(* POU XTEST/Baustein Tests/control_test, CFC *)
PROGRAM control_test
VAR
	Offset : REAL;
	x1: FT_PT1;
	step: REAL;
	t1: TIME := T#1s;
	Out: REAL;
	x2: FT_PT2;
	d: REAL := 0.5;
	out2: REAL;
	x3: FT_PID;
	TV, TN : REAL := 1;
	out3: REAL;
	SET: REAL;
	x4: FT_PI;
	M_in: REAL;
	M_en: BOOL;
	RST: BOOL;
	INTB: REAL := 10;
	KP: REAL := 1;
	KI: REAL := 1;
	L_L: REAL := -1000;
	L_H: REAL := 1000;
	out4: REAL;
	l1: BOOL;
	o1: BOOL;
	l2: BOOL;
	o2: BOOL;
	x5: FT_PT1;
END_VAR
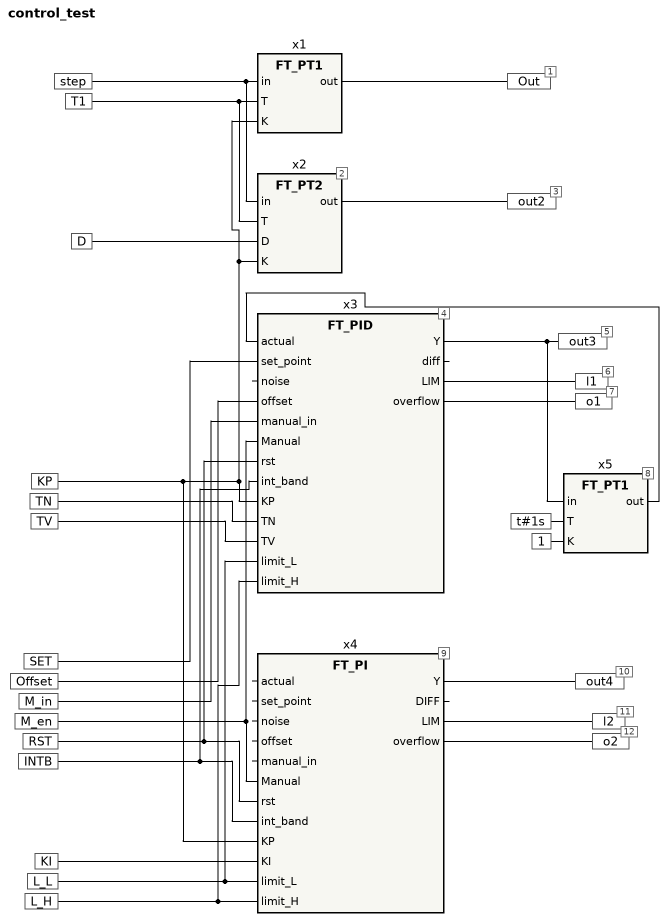
_CFC_ (* Continuous Function Chart, elements in execution order *)
#0 x1:FT_PT1(in: step, T: T1, K: KP)
#1 Out <= #0.out
#2 x2:FT_PT2(in: step, T: T1, D: D, K: KP)
#3 out2 <= #2.out
#4 x3:FT_PID(actual: #8.out, set_point: SET, noise: -, offset: Offset, manual_in: M_in, Manual: M_en, rst: RST, int_band: INTB, KP: KP, TN: TN, TV: TV, limit_L: L_L, limit_H: L_H)
#5 out3 <= #4.Y
#6 l1 <= #4.LIM
#7 o1 <= #4.overflow
#8 x5:FT_PT1(in: #4.Y, T: t#1s, K: 1)
#9 x4:FT_PI(actual: -, set_point: -, noise: -, offset: -, manual_in: -, Manual: M_en, rst: RST, int_band: INTB, KP: KP, KI: KI, limit_L: L_L, limit_H: L_H)
#10 out4 <= #9.Y
#11 l2 <= #9.LIM
#12 o2 <= #9.overflow
_END_CFC_
(* the same logic as Structured Text *)
x1(in := step, T := T1, K := KP);
Out := x1.out;
x2(in := step, T := T1, D := D, K := KP);
out2 := x2.out;
x3(actual := x5.out, set_point := SET, offset := Offset, manual_in := M_in, Manual := M_en, rst := RST, int_band := INTB, KP := KP, TN := TN, TV := TV, limit_L := L_L, limit_H := L_H);
out3 := x3.Y;
l1 := x3.LIM;
o1 := x3.overflow;
x5(in := x3.Y, T := t#1s, K := 1);
x4(Manual := M_en, rst := RST, int_band := INTB, KP := KP, KI := KI, limit_L := L_L, limit_H := L_H);
out4 := x4.Y;
l2 := x4.LIM;
o2 := x4.overflow;
END_PROGRAM

(* POU Engineering/control/FT_PT1, ST *)
FUNCTION_BLOCK FT_PT1
VAR_INPUT
	in : REAL;
	T : TIME;
	K : REAL := 1;
END_VAR
VAR_OUTPUT
	out : REAL;
END_VAR
VAR
	last : DWORD;
	tx: DWORD;
	init: BOOL;
END_VAR

(*
version 1.7	5 jan 2008
programmer 	hugo
tested by		tobias

FT_PT1 is an low pass filter with a programmable time T and faktor K.
 
*)
(* read system time *)
tx := T_PLC_US();

(* startup initialisation *)
IF NOT init THEN
	last := tx;
	init := TRUE;
	out := K * in;
ELSIF T = t#0s THEN
	out := K * in;
ELSE
	out := out + (in * K - out) * (Tx - last) / TIME_TO_REAL(T) * 1E-3;
END_IF;
last := tx;

(*
hm 1.1.2007	rev 1.1
	corrected error while startup value was not correct
	for very small time values real output would run out of range.

hm 3.1.2007	rev 1.2
	corrected an error for falling edge failures.
	added output faktor K.

hm 27. 2. 2007	rev 1.3
	output will be input during init for definitive startup condition.

hm	15.9.2007	rev 1.4
	changed time() to T_PLC_US() for compatibilitxy resons
	increased internal accuracy to Microseconds instead of Milliseconds

hm	23. oct 2007	rev 1.5
	added out := in to the init statements

hm	30. nov 2007	rev 1.6
	changed out to be K * in during initialization

hm	5. jan 2008		rev 1.7
	improved code for better performance
*)
END_FUNCTION_BLOCK

(* POU Engineering/measurements/T_PLC_US, ST *)
FUNCTION T_PLC_US : DWORD
VAR CONSTANT
	debug : BOOL := FALSE;
	N : INT := 0;
	offset : DWORD := 0;
END_VAR
VAR
	tx : TIME;
	temp : DWORD := 1;
END_VAR

(*
version 1.1	12 nov 2007
programmer 	hugo
tested by		tobias

T_PLC_US reads the internal PLC timer and return the time, it has the advantage to be able to set a debug mode 
and speed up the counter to test the plc timer overrun which occurs every 50 days respectively 25 days at siemens S7
this routine also allows to correct the behavior of s7 where the internal plc counter will not count all 32 bits.

*)
tx := TIME();
T_PLC_US := TIME_TO_DWORD(Tx)*1000;
(* hier muss die korrektur für step7 stattfinden
plctime muss den vollen wertebereich von time ausnutzen:
wenn bei step7 time -24tage bis plus 24 tage ist dann muss der timer auch beim überlauf auf -24tage springen 
und auf keinen fall auf 0 !!!!
für siemens muss ein weiterer fb im main eingebunden werden der sicherstellt das alle 32 bits durchgezählt werden.
es kann nur ein fb sein den er muss sich das oberste (32te) bit merken.
oder etwa spring s7 bei überlauf auf -24 tage????? dann wäre keine korrektur nötig.
*)
IF debug THEN
	T_PLC_US := (SHL(T_PLC_US,N) OR SHL(temp,N)-1) + Offset;
END_IF;

(* revision history
hm	14.9.2007	rev 1.0
	original version

hm	12. nov 2007	rev 1.1
	added temporaray variable tx because some compilers could not handle time() as an argument

*)
END_FUNCTION

(* POU Engineering/control/FT_PT2, ST *)
FUNCTION_BLOCK FT_PT2
VAR_INPUT
	in : REAL;
	T : TIME;
	D : REAL;
	K : REAL := 1;
END_VAR
VAR_OUTPUT
	out : REAL;
END_VAR
VAR
	init: BOOL;
	int1 : FT_INT;
	int2 : FT_INT;
	tn: REAL;
END_VAR

(*
version 1.3	30 Nov 2007
programmer 	hugo
tested by		tobias

FT_PT2 is a 2nd grade filter with programmable times T, D and faktor K.
 
*)
(* startup initialisation *)
IF NOT init THEN
	out := K * in;
	init := TRUE;
ELSIF T = t#0s THEN
	out := K * in;
ELSE
	tn := TIME_TO_REAL(T)/1000;
	int1(in := in * K / (TN * TN) - int1.Out * 2 *D / TN - int2.Out / (TN * TN));
	int2(in := int1.Out);
	out := int2.out;
END_IF;

(* revision history

15.1.2007 hm		rev 1.1
	changed formula to new more acurate formula
	old code:
	tx := TIME();
	IF NOT init THEN
		last := tx;
		init := TRUE;
	ELSE
		IF T> t#0s THEN
			out1 := out1 + (in - out1) * TIME_TO_REAL(Tx - last) / TIME_TO_REAL(T);
		ELSE
			out1 := in;
		END_IF;
		IF T > t#0s THEN
			out2 := out2 + (out1 - out2) * TIME_TO_REAL(Tx - last) / TIME_TO_REAL(T);
		ELSE
			out2 := out1;
		END_IF;
		out := out2 * K;
	END_IF;
	last := tx;

hm 		15.9.2007		rev 1.2
	deleted unused code for init system time reading tx	

hm		30.11.2007		rev 1.3
	changed out to be K * in during initialization
	avoind divide by 0 if tn = 0
*)
END_FUNCTION_BLOCK

(* POU Engineering/control/FT_INT, ST *)
FUNCTION_BLOCK FT_INT
VAR_INPUT
	in : REAL;
	K : REAL := 1;
	run : BOOL := 1;
	rst: BOOL := 0;
	out_min : REAL := -1E37;
	out_max : REAL := 1E37;
END_VAR
VAR_OUTPUT
	Out : REAL;
END_VAR
VAR
	last: DWORD;
	in_last : REAL;
	tx: DWORD;
	init: BOOL;
	tc: DWORD;
	out1: REAL;
	out2: REAL;
END_VAR


(*
version 1.8	13. mar 2008
programmer 	hugo
tested by		tobias

FT_int is an integrator with input IN and factor K.
integration is only done while run = true, if run is false integration is stopped and the out remains at the last value.
if run is left unconnected, run is considered true by the function block.
the output ET will display the total integration time from last reset.
a rst input will reset output and the timer ET to 0.
the out_min and out_max values can be set to ,imit the output value range. 
the default for K is 1.

 
*)
(* read and store system time *)
tx := T_PLC_US();
tc := tx - last;

(* startup initialisation *)
IF rst OR NOT init THEN
	out1 := 0;
	out2 := 0;
	init := TRUE;
	last := tx;
ELSIF run AND tc > 0 THEN
	last := tx;
	out1 := out1 + (in + in_last) * tc * K * 5E-7;
	IF ABS(out1) > ABS(out2) THEN
		out2 := out2 + out1;
		out1:= 0;
	END_IF;
ELSIF NOT run THEN
	last := tx;
END_IF;
in_last := in;
out := out1 + out2;
IF out > out_max THEN
	out2 := out_max;
	out1 := 0;
	out := out_max;
ELSIF out < out_min THEN
	out2 := out_min;
	out1 := 0;
	out := out_min;
END_IF;


(*
hm 13.12.2006	rev 1.1
	changed to "trapezregel" which increases accuracy
	before out := out + in * time new: out := out + (in + in_last) / 2 * time

hm 15.1.2007		rev 1.2
	added default for k to be 1.

hm	15.9.2007		rev 1.3
	replaced time() with T_PLC_US for compatibility and performance reason
	increased internal accuracy to microseconds

hm 29. oct 2007		rev 1.4
	changed code so int will not be called is time difference is 0 to increase accuracy on systems
	with cycle times below 1ms

hm	2. dec 2007	 	rev 1.5
	changed code for better performance

hm	5. jan 2008		rev 1.6
	further improvements in performance

hm	8. feb 2008		rev 1.7
	deleted limits +/- 1000 now limit is the range of real
	added variables out1 and out2 to extend the resolution
	corrected an error with elapsed time
	deleted unusfull output ET

hm	13. mar 2008		rev 1.8
	changed preset value out_min to -1e37.
	stop integrator at the limits.
*)
END_FUNCTION_BLOCK

(* POU Engineering/control/FT_PID, ST *)
FUNCTION_BLOCK FT_PID
VAR_INPUT
	actual, set_point, noise, offset, manual_in : REAL;
	Manual : BOOL;
	rst : BOOL := FALSE;
	int_band : REAL := 100;
	KP : REAL := 1.0;
	TN : REAL := 1.0;
	TV : REAL := 1.0;
	limit_L : REAL := -1000;
	limit_H : REAL := 1000;
END_VAR
VAR_INPUT CONSTANT
	int_limit_L : REAL := -1000;
	int_limit_H : REAL := 1000;
END_VAR
VAR_OUTPUT
	Y : REAL;
	diff: REAL;
	LIM, overflow : BOOL;
END_VAR
VAR
	integ : FT_INT;
	deriv : FT_deriv;
END_VAR

(*
version 1.6	5 jan 2008
programmer 	hugo
tested by		tobias

FT_PID is a pid controller with manual functionality.
The PID controller works according to the fomula Y = KP * ( e + 1/TN * INTEG(e) + TV *DERIV(e)) + offset, while e = set_point - actual.
a rst will reset all internal data, while a switch to manual will cause the controller to follow the function Y = manual_in + offset.
limit_h and Limit_l set the possible output range of Y.
the output flags lim will signal that the output limits are active and overflow will signal that the integrator has reached the max or min limit.  

since rev 1.1 the "trapezregel is used for more accuracy.
rev 1.2 added selective integratin which means the integrative component is only active within a small range of the target value 
this avoids the integrator to go to limits while an input setpoint change happened and is only causing overshoots.
the int_band is by default 100 which means the int is active all the time and if set to for example to 0.1 the integrator is only active
while the input is between 0.9 and 1.1 of the set_point value.

default values for KP = 1, TN = 1, TV = 1, LIMIT_L = -1000, LIMIT_H = +1000.
*)
IF NOT rst AND NOT manual THEN
	(* calculate the process error *)
	DIFF := DEAD_BAND(set_point - actual, Noise);
	IF ABS(diff) <= int_band AND NOT overflow AND TN > 0 THEN
		(* integrator is within int_band and needs to be run *)
		integ(in := diff, K := 1/TN, run := TRUE, rst := FALSE, out_min := int_limit_L, out_max := int_limit_H);
		(* check if integrator has reached its limits and set overflow *)
		IF integ.Out >= int_limit_H OR integ.Out <= int_limit_L THEN overflow := TRUE; END_IF;
	ELSE
		(* int_band is exceeded, integrator needs to be cleared *)
		integ(rst := TRUE);
	END_IF;
	(* calculate the derivative part *)
	deriv(in := diff, K := TV);
	(* add up all parts *)
	Y := KP * (integ.Out + deriv.out + diff);
ELSIF rst THEN
	integ(rst := TRUE);		(* reset the integrator *)
	overflow := FALSE;		(* clear the overflow flag *)
	Y := (limit_H + Limit_L) * 0.5 - Offset;	(* set the output between limit_L and limit_L offset will be added again at the end *)
ELSIF manual THEN
	Y := manual_in;
	integ(rst := TRUE);		(* make sure integrator is reset to 0 *)
	overflow := FALSE;		(* manual operation will cancel overflow because integrator was reset *)
END_IF;

(* add offset to Y *)
Y := Y + Offset;

(* limit the outputs and set the lim flag if necessary *)
IF y > limit_H THEN
	y := limit_H;
	lim := TRUE;
ELSIF y < limit_L THEN
	y := limit_L;
	lim := TRUE;
ELSE
	lim := FALSE;
END_IF;


(* old code before rev 1.4
IF rst OR KP = 0 THEN
	y := Offset;
	integ(rst := 1);
	integ.rst := 0;
ELSIF manual THEN
	Y := manual_in + Offset;
	integ(rst := 1);
	integ.rst := 0;
ELSE
	(* calcualtion of the actual PID values *)
	diff := set_point - actual;

	(* integrator is only called if TN > 0 and input is within int_band othewrwise it is disabled *)
	IF TN > 0 AND actual > set_point - int_band AND actual < set_point + int_band THEN
		integ(in := diff, K := 1/TN, out_min := (limit_L - offset) / KP, out_max := (limit_H - offset) / KP);
	ELSE
		integ(rst := 1);
		integ.rst := 0;
	END_IF;
	deriv(in := diff, K := TV);

	(* check if integrator has reached the allowed limits and set overflow if necessary *)
	IF integ.Out >= (limit_H - offset) / KP THEN
		Y := limit_H;
		overflow := TRUE;
	ELSIF integ.Out <= (limit_L - offset) / KP THEN
		Y := limit_L;
		overflow := TRUE;
	ELSE
		Y := KP * (integ.Out + deriv.out + diff) + offset;
		overflow := FALSE;
	END_IF;

	(* this portion limits the output to limit_H and limit_L and set the lim flag if limits are exceeded *)
	IF Y > limit_H THEN
		Y := limit_H;
		Lim := TRUE;
	ELSIF Y < limit_L THEN
		Y := limit_L;
		lim := TRUE;
	ELSE
		lim := FALSE;
	END_IF;
END_IF;
*)

(* revision history

hm 1.12.2006	 	rev 1.1
	changed algorithm to trapezregel for higher accuracy.

hm 3.1.2007		rev 1.2
	added integ_band to select when the integrator is active.

hm	3.3.2007		rev 1.3
	added default values to inputs KP, TN, TV, LIMIT_L und LIMIT_H.

hm 31.oct 2007	rev 1.4
	total rewrite of the module to avoid failures when one of the limits is 0

hm	3.11.2007	rev 1.5
	added noise input to filter noise
	added output diff
	set limit output false when output is within limits
	overfolw was not set correctly

hm	5. jan 2008	rev 1.6
	improved code for better performance
*)
END_FUNCTION_BLOCK

(* POU Engineering/control/FT_deriv, ST *)
FUNCTION_BLOCK FT_deriv
VAR_INPUT
	in : REAL;
	K : REAL := 1;
	run : BOOL := 1;
END_VAR
VAR_OUTPUT
	out : REAL;
END_VAR
VAR
	old: REAL;
	tx: DWORD;
	last: DWORD;
	init: BOOL;
END_VAR


(*
version 1.3	29 oct 2007
programmer 	hugo
tested by		tobias

FT_deriv calculates the derivate over the signal "in" with Faktor "K".
a run input enables or stops the calculation, if left unconnected its true and therfore the calculation is executed.
if K is not specified the default is 1.

*)
(* read system time *)
tx := T_PLC_US();

(* init on firsat startup *)
IF NOT init THEN
	init := TRUE;
	old := in;
	last := tx;
END_IF;
IF run AND tx - last > 0 THEN
	out := (in - old) / DWORD_TO_REAL(tx - last) * 1000000.0 * K;
	last := tx;
ELSE
	out := 0;
	last := tx;
END_IF;
old := in;


(*
hm 3.1.2007			rev 1.1
	added init code for startup
	set the default for K to 1

hm	15. sep 2007	rev 1.2
	replaced Time() with T_PLC_US for compatibility and performance reasons
	increased accuracy and work in microseconds internally

hm 29 oct 2007	rev 1.3
	prohibit calculation when tx - last = 0 to avoid division by 0 and increase accuracy on fast systems
*)
END_FUNCTION_BLOCK

(* POU Engineering/control/DEAD_BAND, ST *)
FUNCTION DEAD_BAND : REAL
VAR_INPUT
	X : REAL;
	L : REAL;
END_VAR
VAR
END_VAR

(*
version 1.0	2 nov 2007
programmer 	hugo
tested by		tobias

DEAD_BAND ist eine lineare Übertragungsfunktion mit Totzone. Die Funktion verschiebt den positiven Teil der Kurve um +L und den negativen Teil der Kurve um -L.
DEAD_BAND = X wenn Abs(X) > L wenn Abs(X) > L
DEAD_BAND = 0 wenn Abs(X) <= L

*)
IF ABS(x) > L THEN
	dead_band := X - sgn(x) * L;
ELSE
	dead_band := 0;
END_IF;

(* revision history
hm		2.11.07	rev 1.0
	original version
*)
END_FUNCTION

(* POU Engineering/control/FT_PI, ST *)
FUNCTION_BLOCK FT_PI
VAR_INPUT
	actual, set_point, noise, offset, manual_in : REAL;
	Manual : BOOL;
	rst : BOOL := FALSE;
	int_band : REAL := 100;
	KP : REAL := 1.0;
	KI : REAL := 1.0;
	limit_L : REAL := -1000;
	limit_H : REAL := 1000;
END_VAR
VAR_INPUT CONSTANT
	int_limit_L : REAL := -1000;
	int_limit_H : REAL := 1000;
END_VAR
VAR_OUTPUT
	Y : REAL;
	DIFF : REAL;
	LIM, overflow : BOOL;
END_VAR
VAR
	integ : FT_INT;
END_VAR

(*
version 1.2	5 jan 2008
programmer 	hugo
tested by		tobias

FT_PI is a PI controller with manual functionality.
The PID controller works according to the fomula Y = e *(KP+ KI * INTEG(e) ) + offset, while e = set_point - actual.
a rst will reset all internal data, while a switch to manual will cause the controller to follow the function Y = manual_in + offset.
limit_h and Limit_l set the possible output range of Y.
the output flags lim will signal that the output limits are active and overflow will signal that the integrator has reached its limits.

since rev 1.1 the "trapezregel is used for more accuracy.
rev 1.2 added selective integratin which means the integrative component is only active within a small range of the target value 
this avoids the integrator to go to limits while an input setpoint change happened and is only causing overshoots.
the int_band is by default 100 which means the int is active all the time and if set to for example to 0.1 the integrator is only active
while the input is between 0.9 and 1.1 of the set_point value.

default values for KP = 1, TN = 1, TV = 1, LIMIT_L = -1000, LIMIT_H = +1000.
*)
IF NOT rst AND NOT manual THEN
	(* calculate the process error *)
	DIFF := dead_band(set_point - actual, Noise);
	IF ABS(diff) <= int_band AND NOT overflow THEN
		(* integrator is within int_band and needs to be run *)
		integ(in := diff, K := KI, run := TRUE, rst := FALSE, out_min := int_limit_L, out_max := int_limit_H);
		(* check if integrator has reached its limits and set overflow *)
		IF integ.Out >= int_limit_H OR integ.Out <= int_limit_L THEN overflow := TRUE; END_IF;
	ELSE
		(* int_band is exceeded, integrator needs to be cleared *)
		integ(rst := TRUE);
	END_IF;
	Y := KP * diff + integ.Out;
ELSIF rst THEN
	integ(rst := TRUE);		(* reset the integrator *)
	overflow := FALSE;		(* clear the overflow flag *)
	Y := (limit_H + Limit_L) * 0.5 - Offset;	(* set the output between limit_L and limit_L offset will be added again at the end *)
ELSIF manual THEN
	Y := manual_in;
	integ(rst := TRUE);		(* make sure integrator is reset to 0 *)
	overflow := FALSE;		(* manual operation will cancel overflow because integrator was reset *)
END_IF;

(* add offset to Y *)
Y := Y + Offset;

(* limit the outputs and set the lim flag if necessary *)
IF y > limit_H THEN
	y := limit_H;
	lim := TRUE;
ELSIF y < limit_L THEN
	y := limit_L;
	lim := TRUE;
ELSE
	lim := FALSE;
END_IF;



(* revision history
hm 	31.10.2007 	rev 1.0
	original version

hm	3.11.2007	rev 1.1
	added noise input to filter noise
	added output diff
	set limit output false when output is within limits
	overfolw was not set correctly

hm	5. jan 2008	rev 1.2
	improved performance
*)
END_FUNCTION_BLOCK

(* POU XTEST/Baustein Tests/crc_test, CFC *)
PROGRAM crc_test
VAR
	arr : ARRAY[1..9] OF BYTE := 49, 50, 51, 52, 53, 54, 55, 56, 57;
	code: DWORD;
	hex: STRING;
END_VAR
VAR (* helpers for the ST form of the networks *)
	_t1 : DWORD;
END_VAR
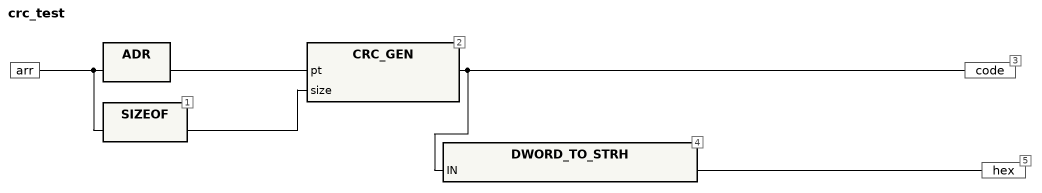
_CFC_ (* Continuous Function Chart, elements in execution order *)
#0 ADR(arr)
#1 SIZEOF(arr)
#2 CRC_GEN(pt: #0, size: #1, Polynom_L := 263, init := 255, XOR_out := 255, rev_in := TRUE, rev_out := TRUE)
#3 code <= #2
#4 DWORD_TO_STRH(IN: #2)
#5 hex <= #4
_END_CFC_
(* the same logic as Structured Text *)
_t1 := CRC_GEN(ADR(arr), SIZEOF(arr));
code := _t1;
hex := DWORD_TO_STRH(IN := _t1);
END_PROGRAM

(* POU String/CODE, ST *)
FUNCTION CODE : BYTE
VAR_INPUT
	STR : STRING;
	POS : INT;
END_VAR
VAR
	PT : POINTER TO BYTE;
END_VAR

(*
version 1.0	9. mar. 2008
programmer 	hugo
tested by		tobias

code extracts the code of a character at position POS of a string STR.

*)
IF pos < 1 OR pos > LEN(str) THEN
	CODE := 0;
	RETURN;
ELSE
	PT := ADR(STR) + INT_TO_DWORD(pos - 1);
	CODE := pt^;
END_IF;

(* revision history
hm		9. mar. 2008		rev 1.0
	original version

*)
END_FUNCTION

(* POU Logic/Others/CRC_GEN, ST *)
FUNCTION CRC_GEN : DWORD

VAR_INPUT
	pt : POINTER TO ARRAY[0..32000] OF BYTE;
	size : INT;
END_VAR
VAR_INPUT CONSTANT
	Polynom_L : DWORD;
	Polynom_32 : BOOL;
	init: DWORD := 0;
	XOR_out : DWORD;
	rev_in : BOOL;
	rev_out : BOOL;
END_VAR
VAR
	polynom : DWORD;
	p_length : INT;
	BS : BYTE;
	data : DWORD;
	count : BYTE;
	temp : BOOL;
	step: INT;
	s4: INT;
END_VAR

(*
version 1.3	2 jan 2008
programmer 	hugo
tested by		tobias

CRC_GEN generates a CRC checksum from a block of data and returns  the checksum in a DWORD to be connected to the data for transmission.
the CRC Polynom is specified with the config variable Polynom_L which holds the lowest 32 bits of the polynom and Polynom_33 which holds bit 33 of the Polynom.
A Polynom x4 + X + 1 is represented by 10011.
The input data is an array of byte of any size, the function is called by CRC_GEN(ADR(array),SIZEOF(array)).

*)
(* check for polynom length and calculate p_length polynom will be aligned to high side of word*)
polynom := polynom_L;
IF polynom_32 THEN
	p_length := 33;
ELSE;
	p_length := 32;
	WHILE p_length > 0 AND NOT polynom.31 DO
		p_length := p_length - 1;
		Polynom := SHL(polynom,1);
	END_WHILE;
	Polynom := SHL(polynom,1);
END_IF;


(* load start code and first data byte for crc calculation *)
data := init;
IF rev_in THEN bs := reverse(pt^[0]); ELSE bs := pt^[0]; END_IF;

(* calcualte checksum *)
s4 := size + 4;
WHILE step < s4 DO
	temp := data.31;
	data := SHL(data,1);
	data.0 := BS.7;
	bs := SHL(bs,1);
	count := count + 1;
	IF count = 8 THEN
		step := step + 1;
		count := 0;
		IF step < size THEN
			IF rev_in THEN bs := reverse(pt^[step]); ELSE bs := pt^[step]; END_IF;
		END_IF;
	END_IF;
	(* check highest bit if true then xor polynom *)
	IF temp THEN data := data XOR polynom; END_IF;
END_WHILE;

(* reverse crc if necessary *)
IF rev_out THEN
	CRC_GEN.31 := data.31;
	FOR step := p_length TO 3 BY -1 DO
		data := SHL(data,1);
		CRC_GEN := SHR(CRC_GEN,1);
		CRC_GEN.31 := data.31;
	END_FOR;
ELSE
	CRC_GEN := data;
END_IF;

(* final XOR and align crc checksum to right side of dword *)
CRC_GEN := CRC_GEN XOR SHL(xor_out, 33 - p_length);
CRC_GEN := SHR(CRC_GEN,33 - p_length);


(* old code prior to rev 1.2
B1 := pt^[0];
IF size > 1 THEN B2 := pt^[1]; ELSE B2 := 0; END_IF;
IF size > 2 THEN B3 := pt^[2]; ELSE B3 := 0; END_IF;
IF size > 3 THEN B4 := pt^[3]; ELSE B4 := 0; END_IF;
IF size > 4 THEN BS := pt^[4]; ELSE BS := 0; END_IF;
data := DWord_of_Byte(B4,B3,B2,B1);

WHILE step < size DO
	temp := data.31;
	data := SHL(data,1);
	data.0 := BS.7;
	bs := SHL(bs,1);
	count := count + 1;
	IF count = 8 THEN
		step := step + 1;
		count := 0;
		IF step + 4 < size THEN bs := pt^[step+ 4]; END_IF;
	END_IF;
	(* check highest bit if true then xor polynom *)
	IF temp = TRUE THEN
		data := data XOR polynom;
	END_IF;
END_WHILE;

(* align crc checksum to right side of dword *)
CRC_GEN := SHR(data,32 - p_length +1);
*)


(* typical crc polynoms

CRC-4-ITU 			x4 + x + 1 					(ITU G.704, p. 12) 	0x3 or 0xC (0x9)
CRC-5-ITU 			x5 + x4 + x2 + 1 			(ITU G.704, p. 9) 	0x15 or 0x15 (0x0B) Bluetooth
CRC-5-USB 			x5 + x2 + 1 				(use: USB token packets) 	0x05 or 0x14 (0x9)
CRC-6-ITU 			x6 + x + 1 					(ITU G.704, p. 3) 	0x03 or 0x30 (0x21)
CRC-7 				x7 + x3 + 1 				(use: telecom systems, MMC) 	0x09 or 0x48 (0x11)
CRC-8-ATM 			x8 + x2 + x + 1 				(use: ATM HEC) 	0x07 or 0xE0 (0xC1)
CRC-8-CCITT 		x8 + x7 + x3 + x2 + 1 		(use: 1-Wire bus) 	0x8D or 0xB1 (0x63)
CRC-8-Dallas/Maxim 	x8 + x5 + x4 + 1 			(use: 1-Wire bus) 	0x31 or 0x8C (0x19)
CRC-8 				x8 + x7 + x6 + x4 + x2 + 1 	0xD5 or 0xAB (0x57)
CRC-8-SAE J1850 	x8 + x4 + x3 + x2 + 1 		0x1D or 0xB8
CRC-10 				x10 + x9 + x5 + x4 + x + 1 	0x233 or 0x331 (0x263)
CRC-12 				x12 + x11 + x3 + x2 + x + 1 (use: telecom systems) 	0x80F or 0xF01 (0xE03)
CRC-15-CAN 			x15 + x14 + x10 + x8 + x7 + x4 + x3 + 1 	0x4599 or 0x4CD1 (0x19A3)
CRC-16-Fletcher 	Not a CRC; see Fletcher's checksum 	Used in Adler-32 A & B CRCs
CRC-16-CCITT 	x16 + x12 + x5 + 1 (XMODEM,X.25, V.41, Bluetooth, PPP, IrDA; known as "CRC-CCITT") 	0x1021 or 0x8408 (0x0811)
CRC-16-IBM 	x16 + x15 + x2 + 1 (USB, many others; also known as "CRC-16") 	0x8005 or 0xA001 (0x4003)
CRC-24-Radix-64 	x24 + x23 + x18 + x17 + x14 + x11 + x10 + x7 + x6 + x5 + x4 + x3 + x + 1 	0x864CFB or 0xDF3261 (0xBE64C3)
CRC-32-Adler 	Not a CRC; see Adler-32 	See Adler-32
CRC-32-MPEG2 	x32 + x26 + x23 + x22 + x16 + x12 + x11 + x10 + x8 + x7 + x5 + x4 + x2 + x + 1 	0x04C11DB7 or 0xEDB88320 (0xDB710641) Also used in IEEE 802.3
CRC-32-IEEE 802.3 	x32 + x26 + x23 + x22 + x16 + x12 + x11 + x10 + x8 + x7 + x5 + x4 + x2 + x + 1 (V.42) 	0x04C11DB7 or 0xEDB88320 (0xDB710641)
CRC-32C (Castagnoli) 	x32 + x28 + x27 + x26 + x25 + x23 + x22 + x20 + x19 + x18 + x14 + x13 + x11 + x10 + x9 + x8 + x6 + 1 	0x1EDC6F41 or 0x82F63B78 (0x05EC76F1)
CRC-64-ISO 	x64 + x4 + x3 + x + 1 (use: ISO 3309) 	0x000000000000001B or 0xD800000000000000 (0xB000000000000001)
CRC-64-ECMA-182 	x64 + x62 + x57 + x55 + x54 + x53 + x52 + x47 + x46 + x45 + x40 + x39 + x38 + x37 + x35 + x33 + x32 + x31 + x29 + x27 + x24 + x23 + x22 + x21 + x19 + x17 + x13 + x12 + x10 + x9 + x7 + x4 + x + 1
(as described in ECMA-182 p.63) 	0x42F0E1EBA9EA3693 or 0xC96C5795D7870F42 (0x92D8AF2BAF0E1E85)

*)

(* revision history

hm		9.6.2007	rev 1.0		
	original version 

hm		11.9.2007	rev 1.1
	deleted unused variable i

hm		9. oct 2007 rev 1.2
	added init code for crc and xor_out
	added refelct in and reflect_out (rev_in und Rev_out)

hm		2. jan 2008	rev 1.3
	small changes for performance improvements
*)
END_FUNCTION

(* POU Logic/gate logic/reverse, ST *)
FUNCTION reverse : BYTE
VAR_INPUT
	IN : BYTE;
END_VAR
VAR
END_VAR

(*
	version 1.1	18. feb 2008
	programmer 	hugo
	tested BY		tobias

This function reverses the bits of a byte so that after execution bit 7 is at bit 0 location and so forth.

*)
reverse := SHL(in,7) OR SHR(in,7) OR (ROR(in,3) AND 2#01000100) OR (ROL(in,3) AND 2#00100010)
	OR (SHL(in,1) AND 2#00010000) OR (SHR(in,1) AND 2#00001000);


(* revision history
hm		9.oct 2007		rev 1.0
	original version

hm		18. feb 2008	rev 1.1
	improved performance
*)
END_FUNCTION

(* POU String/DWORD_TO_STRH, ST *)
FUNCTION DWORD_TO_STRH : STRING
VAR_INPUT
	IN : DWORD;
END_VAR
VAR
	i : INT;
	temp : BYTE;
	pt : POINTER TO BYTE;
END_VAR

(*
version 1.2	15 dec 2007
programmer 	hugo
tested by		tobias

DWORD_TO_STRINGH converts a DWORD to a String of Hexadecimal represented by '0' .. '9' and 'A' .. 'F'.
The lowest order Character will be on the right and the high order Character on the left.

*)
(* read output adress to pointer *)
pt := ADR(DWORD_TO_STRH) + 8;
(* wirte the closing byte for the string *)
pt^:= 0;

(* write the 8 hex characters backwards *)
FOR i := 1 TO 8 DO;
	(* decrement the pointer *)
	pt := pt - 1;
	(* read the lowest order hex value *)
	temp := DWORD_TO_BYTE(in AND 16#0000000F);
	(* convert value to hex character *)
	IF temp <= 9 THEN temp := temp + 48; ELSE temp := temp + 55; END_IF;
	(* write character to output string *)
	PT^ := temp;
	(* shift in for nect hex character *)
	in := SHR(in,4);
END_FOR;


(* code beofre rev 1.2
FOR i := 1 TO 8 DO
	X := DWORD_TO_BYTE(in AND 2#1111);
	IF X <= 9 THEN X := X + 48; ELSE X := X + 55; END_IF;
	Cx := CHR(X);
	temp := CONCAT(Cx, temp);
	in := SHR(in,4);
END_FOR;
DWORD_TO_STRH := temp;
*)


(* revision history
hm		9.6.2007		rev 1.0		
	original version 

hm		11.9.2007		rev 1.1
	changed coding for compatibility with twincat, concat cannot support a function as an argument.

hm		15.12.2007		rev 1.2
	changed code for better performance
*)
END_FUNCTION

(* POU XTEST/Baustein Tests/esr_test, CFC *)
PROGRAM esr_test
VAR
	x1: ESR_collect;
	eout  : ARRAY[0..63] OF esr_data;
	x2: ESR_MON_B8;
	e0, e1, e2, e3, e4, e5, e6, e7: BOOL;
	dtime: DT;
	x3: ESR_MON_R4;
	r0, r1, r2, r3: REAL;
	x4: ESR_MON_X8;
	b0, b1, b2, b3, b4, b5, b6, b7: BYTE;
	m: BYTE;
	n: INT;
END_VAR
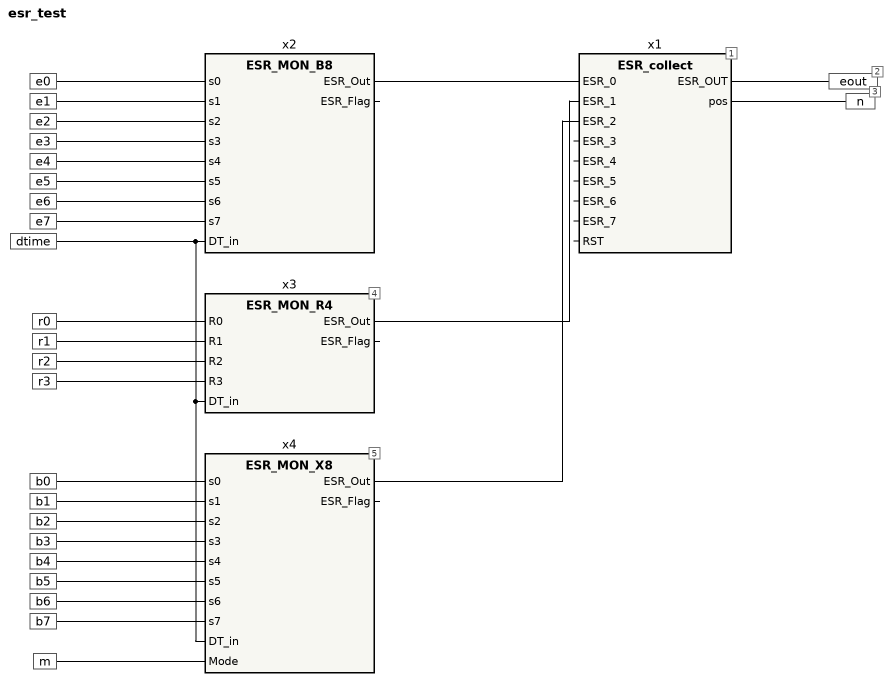
_CFC_ (* Continuous Function Chart, elements in execution order *)
#0 x2:ESR_MON_B8(s0: e0, s1: e1, s2: e2, s3: e3, s4: e4, s5: e5, s6: e6, s7: e7, DT_in: dtime, a0 := 'binär 0', a1 := 'binär 1', a2 := 'binär 2', a3 := 'binär 3', a4 := 'binär 4', a5 := 'binär 5', a6 := 'binär 6', a7 := 'binär 7')
#1 x1:ESR_collect(ESR_0: #0.ESR_Out, ESR_1: #4.ESR_Out, ESR_2: #5.ESR_Out, ESR_3: -, ESR_4: -, ESR_5: -, ESR_6: -, ESR_7: -, RST: -)
#2 eout <= #1.ESR_OUT
#3 n <= #1.pos
#4 x3:ESR_MON_R4(R0: r0, R1: r1, R2: r2, R3: r3, DT_in: dtime, a0 := 'real 0', a1 := 'real 1', a2 := 'real 2', a3 := 'real 3', s0 := 0.0, s1 := 0.1, s2 := 0.2, s3 := 0.3)
#5 x4:ESR_MON_X8(s0: b0, s1: b1, s2: b2, s3: b3, s4: b4, s5: b5, s6: b6, s7: b7, DT_in: dtime, Mode: m, a0 := 'status 0', a1 := 'status 1', a2 := 'status 2', a3 := 'status 3', a4 := 'status 4', a5 := 'status 5', a6 := 'status 6', a7 := 'status 7')
_END_CFC_
(* the same logic as Structured Text *)
x2(s0 := e0, s1 := e1, s2 := e2, s3 := e3, s4 := e4, s5 := e5, s6 := e6, s7 := e7, DT_in := dtime, a0 := 'binär 0', a1 := 'binär 1', a2 := 'binär 2', a3 := 'binär 3', a4 := 'binär 4', a5 := 'binär 5', a6 := 'binär 6', a7 := 'binär 7');
x1(ESR_0 := x2.ESR_Out, ESR_1 := x3.ESR_Out, ESR_2 := x4.ESR_Out);
eout := x1.ESR_OUT;
n := x1.pos;
x3(R0 := r0, R1 := r1, R2 := r2, R3 := r3, DT_in := dtime, a0 := 'real 0', a1 := 'real 1', a2 := 'real 2', a3 := 'real 3', s0 := 0.0, s1 := 0.1, s2 := 0.2, s3 := 0.3);
x4(s0 := b0, s1 := b1, s2 := b2, s3 := b3, s4 := b4, s5 := b5, s6 := b6, s7 := b7, DT_in := dtime, Mode := m, a0 := 'status 0', a1 := 'status 1', a2 := 'status 2', a3 := 'status 3', a4 := 'status 4', a5 := 'status 5', a6 := 'status 6', a7 := 'status 7');
END_PROGRAM

(* POU Other/ESR_collect, ST *)
FUNCTION_BLOCK ESR_collect
VAR_INPUT
	ESR_0, ESR_1, ESR_2, ESR_3, ESR_4, ESR_5, ESR_6, ESR_7 : ARRAY [0..3] OF esr_data;
	RST : BOOL;
END_VAR
VAR_OUTPUT
	ESR_OUT : ARRAY[0..63] OF esr_data;
	pos : INT;
END_VAR
VAR CONSTANT
	max_in : INT := 3; (* maximum element of input variable *)
	max_out : INT := 63; (* maximum element of output array *)
END_VAR
VAR
	cnt : INT;
END_VAR

(*
version 1.0	26 jan 2007
programmer 	hugo
tested by		tobias

ESR_collect collects esr data from up to 8 esr_mon modules and stroes them in an output array.
the output pos will display the position of the last element in the array.
if the array will be full, the oldest element is overwritten.

*)
IF rst THEN
	pos := 0;
	FOR cnt := 0 TO 63 DO
		esr_out[cnt].typ := 0;
		esr_out[cnt].adress := '';
		esr_out[cnt].DS := DT#1970-1-1-00:00;
		esr_out[cnt].TS := T#0ms;
		esr_out[cnt].data[0] := 0;
		esr_out[cnt].data[1] := 0;
		esr_out[cnt].data[2] := 0;
		esr_out[cnt].data[3] := 0;
		esr_out[cnt].data[4] := 0;
		esr_out[cnt].data[5] := 0;
		esr_out[cnt].data[6] := 0;
		esr_out[cnt].data[7] := 0;
	END_FOR;
ELSE
	FOR cnt := 0 TO max_in DO
		IF esr_0[cnt].typ > 0 THEN
			esr_out[pos] := esr_0[cnt];
			pos := pos + 1;
			IF pos > max_out THEN pos := 0; END_IF;
		END_IF;
	END_FOR;
	FOR cnt := 0 TO max_in DO
		IF esr_1[cnt].typ > 0 THEN
			esr_out[pos] := esr_1[cnt];
			pos := pos + 1;
			IF pos > max_out THEN pos := 0; END_IF;
		END_IF;
	END_FOR;
	FOR cnt := 0 TO max_in DO
		IF esr_2[cnt].typ > 0 THEN
			esr_out[pos] := esr_2[cnt];
			pos := pos + 1;
			IF pos > max_out THEN pos := 0; END_IF;
		END_IF;
	END_FOR;
	FOR cnt := 0 TO max_in DO
		IF esr_3[cnt].typ > 0 THEN
			esr_out[pos] := esr_3[cnt];
			pos := pos + 1;
			IF pos > max_out THEN pos := 0; END_IF;
		END_IF;
	END_FOR;
	FOR cnt := 0 TO max_in DO
		IF esr_4[cnt].typ > 0 THEN
			esr_out[pos] := esr_4[cnt];
			pos := pos + 1;
			IF pos > max_out THEN pos := 0; END_IF;
		END_IF;
	END_FOR;
	FOR cnt := 0 TO max_in DO
		IF esr_5[cnt].typ > 0 THEN
			esr_out[pos] := esr_5[cnt];
			pos := pos + 1;
			IF pos > max_out THEN pos := 0; END_IF;
		END_IF;
	END_FOR;
	FOR cnt := 0 TO max_in DO
		IF esr_6[cnt].typ > 0 THEN
			esr_out[pos] := esr_6[cnt];
			pos := pos + 1;
			IF pos > max_out THEN pos := 0; END_IF;
		END_IF;
	END_FOR;
	FOR cnt := 0 TO max_in DO
		IF esr_7[cnt].typ > 0 THEN
			esr_out[pos] := esr_7[cnt];
			pos := pos + 1;
			IF pos > max_out THEN pos := 0; END_IF;
		END_IF;
	END_FOR;
END_IF;

(* revision history
hm	26.jan 2007		rev 1.0
	original version

hm	8. dec 2007		rev 1.1
	added reset input

*)
END_FUNCTION_BLOCK

(* POU Other/ESR_MON_B8, ST *)
FUNCTION_BLOCK ESR_MON_B8
VAR_INPUT
	s0, s1, s2, s3, s4, s5, s6, s7 : BOOL;
	DT_in : DT;
END_VAR
VAR_INPUT CONSTANT
	a0, a1, a2, a3, a4, a5, a6, a7 : STRING(10);
END_VAR
VAR_OUTPUT
	ESR_Out: ARRAY [0..3] OF esr_data;
	ESR_Flag : BOOL;
END_VAR
VAR
	x0, x1, x2, x3, x4, x5, x6, x7 : BOOL;
	tx: TIME;
	cnt : INT;
END_VAR

(*
version 1.1	17 sep 2007
programmer 	hugo
tested by		tobias

ESR_mon_B8 monitores up to 8 binary inputs and reports changes with time stamd and adress label.
the module checks 8 inputs for a change and reports all changes with time and adress stamp to the output.
4 events maximum can be collected at once within the same cycle

*)
(* read system timer *)
tx := DWORD_TO_TIME(T_PLC_MS());

ESR_Flag := FALSE;
esr_out[3].typ := 0;
esr_out[2].typ := 0;
esr_out[1].typ := 0;
esr_out[0].typ := 0;
cnt := 0;

(* check if inputs have chaged and fill buffer *)
IF s0 <> X0 THEN
	IF s0 THEN esr_out[cnt].typ := 11; ELSE 	esr_out[cnt].typ := 10; END_IF;
	esr_out[cnt].adress := a0;
	esr_out[cnt].DS := DT_in;
	esr_out[cnt].TS := TX;
	X0 := S0;
	cnt := cnt + 1;
	esr_flag := TRUE;
END_IF;
IF s1 <> X1 THEN
	IF s1 THEN esr_out[cnt].typ := 11; ELSE 	esr_out[cnt].typ := 10; END_IF;
	esr_out[cnt].adress := a1;
	esr_out[cnt].DS := DT_in;
	esr_out[cnt].TS := TX;
	X1 := S1;
	cnt := cnt + 1;
	esr_flag := TRUE;
END_IF;
IF s2 <> X2 THEN
	IF s2 THEN esr_out[cnt].typ := 11; ELSE 	esr_out[cnt].typ := 10; END_IF;
	esr_out[cnt].adress := a2;
	esr_out[cnt].DS := DT_in;
	esr_out[cnt].TS := TX;
	X2 := S2;
	cnt := cnt + 1;
	esr_flag := TRUE;
END_IF;
IF s3 <> X3 THEN
	IF s3 THEN esr_out[cnt].typ := 11; ELSE 	esr_out[cnt].typ := 10; END_IF;
	esr_out[cnt].adress := a3;
	esr_out[cnt].DS := DT_in;
	esr_out[cnt].TS := TX;
	X3 := S3;
	cnt := cnt + 1;
	esr_flag := TRUE;
END_IF;
IF s4 <> X4 AND cnt < 4 THEN
	IF s4 THEN esr_out[cnt].typ := 11; ELSE 	esr_out[cnt].typ := 10; END_IF;
	esr_out[cnt].adress := a4;
	esr_out[cnt].DS := DT_in;
	esr_out[cnt].TS := TX;
	X4 := S4;
	cnt := cnt + 1;
	esr_flag := TRUE;
END_IF;
IF s5 <> X5  AND cnt < 4 THEN
	IF s5 THEN esr_out[cnt].typ := 11; ELSE 	esr_out[cnt].typ := 10; END_IF;
	esr_out[cnt].adress := a5;
	esr_out[cnt].DS := DT_in;
	esr_out[cnt].TS := TX;
	X5 := S5;
	cnt := cnt + 1;
	esr_flag := TRUE;
END_IF;
IF s6 <> X6  AND cnt < 4 THEN
	IF s6 THEN esr_out[cnt].typ := 11; ELSE 	esr_out[cnt].typ := 10; END_IF;
	esr_out[cnt].adress := a6;
	esr_out[cnt].DS := DT_in;
	esr_out[cnt].TS := TX;
	X6 := S6;
	cnt := cnt + 1;
	esr_flag := TRUE;
END_IF;
IF s7 <> X7  AND cnt < 4 THEN
	IF s7 THEN esr_out[cnt].typ := 11; ELSE 	esr_out[cnt].typ := 10; END_IF;
	esr_out[cnt].adress := a7;
	esr_out[cnt].DS := DT_in;
	esr_out[cnt].TS := TX;
	X7 := S7;
	cnt := cnt + 1;
	esr_flag := TRUE;
END_IF;

(* revision history
hm	26. jan 2007		rev 1.0
	original version

hm	17. sep 2007	rev 1.1
	replaced time() with T_PLC_MS() for compatibility reasons
	
*)
END_FUNCTION_BLOCK

(* POU Other/ESR_MON_R4, ST *)
FUNCTION_BLOCK ESR_MON_R4
VAR_INPUT
	R0, R1, R2, R3 : REAL;
	DT_in : DT;
END_VAR
VAR_INPUT CONSTANT
	a0, a1, a2, a3 : STRING(10);
	s0, s1, s2, s3 : REAL;
END_VAR
VAR_OUTPUT
	ESR_Out: ARRAY [0..3] OF esr_data;
	ESR_Flag : BOOL;
END_VAR
VAR
	p0, p1, p2, p3 : POINTER TO DWORD;
	x0, x1, x2, x3 : REAL;
	tx: TIME;
	cnt : INT;
END_VAR

(*
version 1.2 8 dec 2007
programmer 	hugo
tested by		tobias

ESR_mon_R4 monitores up to 4 Real inputs and reports changes with time stamd and adress label.
the module checks 4 inputs for a change of more than the specified sensitivity S and reports all changes with time and adress stamp to the output.

*)
(* read system timer *)
tx := DWORD_TO_TIME(T_PLC_MS());
P0 := ADR(R0);
P1 := ADR(R1);
P2 := ADR(R2);
P3 := ADR(R3);

ESR_Flag := FALSE;
esr_out[3].typ := 0;
esr_out[2].typ := 0;
esr_out[1].typ := 0;
esr_out[0].typ := 0;
cnt := 0;

(* check if inputs have chaged and fill buffer *)
IF differ(R0,  X0, S0) THEN
	esr_out[cnt].typ := 20;
	esr_out[cnt].adress := a0;
	esr_out[cnt].DS := DT_in;
	esr_out[cnt].TS := TX;
	esr_out[cnt].data[0] := Byte_of_Dword(REAL_TO_DWORD(P0^),0);
	esr_out[cnt].data[1] := Byte_of_Dword(REAL_TO_DWORD(P0^),1);
	esr_out[cnt].data[2] := Byte_of_Dword(REAL_TO_DWORD(P0^),2);
	esr_out[cnt].data[3] := Byte_of_Dword(REAL_TO_DWORD(P0^),3);
	X0 := R0;
	cnt := cnt + 1;
	esr_flag := TRUE;
END_IF;
IF differ(R1,  X1, S1) THEN
	esr_out[cnt].typ := 20;
	esr_out[cnt].adress := a1;
	esr_out[cnt].DS := DT_in;
	esr_out[cnt].TS := TX;
	esr_out[cnt].data[0] := Byte_of_Dword(REAL_TO_DWORD(P1^),0);
	esr_out[cnt].data[1] := Byte_of_Dword(REAL_TO_DWORD(P1^),1);
	esr_out[cnt].data[2] := Byte_of_Dword(REAL_TO_DWORD(P1^),2);
	esr_out[cnt].data[3] := Byte_of_Dword(REAL_TO_DWORD(P1^),3);
	X1 := R1;
	cnt := cnt + 1;
	esr_flag := TRUE;
END_IF;
IF differ(R2,  X2, S2) THEN
	esr_out[cnt].typ := 20;
	esr_out[cnt].adress := a2;
	esr_out[cnt].DS := DT_in;
	esr_out[cnt].TS := TX;
	esr_out[cnt].data[0] := Byte_of_Dword(REAL_TO_DWORD(P2^),0);
	esr_out[cnt].data[1] := Byte_of_Dword(REAL_TO_DWORD(P2^),1);
	esr_out[cnt].data[2] := Byte_of_Dword(REAL_TO_DWORD(P2^),2);
	esr_out[cnt].data[3] := Byte_of_Dword(REAL_TO_DWORD(P2^),3);
	X2 := R2;
	cnt := cnt + 1;
	esr_flag := TRUE;
END_IF;
IF differ(R3,  X3, S3) THEN
	esr_out[cnt].typ := 20;
	esr_out[cnt].adress := a3;
	esr_out[cnt].DS := DT_in;
	esr_out[cnt].TS := TX;
	esr_out[cnt].data[0] := Byte_of_Dword(REAL_TO_DWORD(P3^),0);
	esr_out[cnt].data[1] := Byte_of_Dword(REAL_TO_DWORD(P3^),1);
	esr_out[cnt].data[2] := Byte_of_Dword(REAL_TO_DWORD(P3^),2);
	esr_out[cnt].data[3] := Byte_of_Dword(REAL_TO_DWORD(P3^),3);
	X3 := R3;
	cnt := cnt + 1;
	esr_flag := TRUE;
END_IF;


(* revision history
hm	26. jan 2007	rev 1.0
	original version

hm	17. sep 2007	rev 1.1
	replaced time() with T_PLC_MS() for compatibility reasons

hm	8 dec 2007		rev 1.2
	corrected an error while esr typ would not be set
*)
END_FUNCTION_BLOCK

(* POU Logic/gate logic/Byte_of_Dword, ST *)
FUNCTION Byte_of_Dword : BYTE
VAR_INPUT
	in : DWORD;
	N : BYTE;
END_VAR
VAR
END_VAR

(*
version 1.1	2 jan 2008
programmer 	hugo
tested by		tobias

this function extracts a single byte from the nth position from right (right is lowest byte) 
the lower byte (starting with Bit0 from in) is selected with N=0.
*)
Byte_of_Dword := DWORD_TO_BYTE(SHR(in,n*8));

(* revision history
hm	17. jan 2007	rev 1.0
	original version

hm	2. jan 2008		rev 1.1
	improved performance

*)
END_FUNCTION

(* POU Other/ESR_MON_X8, ST *)
FUNCTION_BLOCK ESR_MON_X8
VAR_INPUT
	s0, s1, s2, s3, s4, s5, s6, s7 : BYTE;
	DT_in : DT;
	Mode : BYTE := 3;
END_VAR
VAR_INPUT CONSTANT
	a0, a1, a2, a3, a4, a5, a6, a7 : STRING(10);
END_VAR
VAR_OUTPUT
	ESR_Out: ARRAY [0..3] OF esr_data;
	ESR_Flag : BOOL;
END_VAR
VAR
	x0, x1, x2, x3, x4, x5, x6, x7 : BYTE;
	tx: TIME;
	cnt : INT;
END_VAR

(*
version 1.1	17 sep 2007
programmer 	hugo
tested by		tobias

ESR_MON_X8 is a status and error collector.
the module checks 8 status inputs for a change and reports up to 4 input changes with time and adress stamp to the output.
the mode can be 
1 for error only
2 for error and status
3 for error, status and debug
the adress label of the 8 inputs can be configured individually.
*)
(* read system timer *)
tx := DWORD_TO_TIME(T_PLC_MS());

ESR_Flag := FALSE;
esr_out[3].typ := 0;
esr_out[2].typ := 0;
esr_out[1].typ := 0;
esr_out[0].typ := 0;
cnt := 0;

(* check if inputs have chaged and fill buffer *)
IF s0 <> X0 AND ((s0 < 100) OR (S0 > 99 AND S0 < 200 AND mode >= 2) OR (S0 > 199 AND mode = 3)) THEN
	esr_out[cnt] := status_to_ESR(s0, a0, DT_in, TX);
	X0 := S0;
	cnt := cnt + 1;
	esr_flag := TRUE;
END_IF;
IF s1 <> X1 AND ((s1 < 100) OR (S1 > 99 AND S1 < 200 AND mode >= 2) OR (S1 > 199 AND mode = 3)) THEN
	esr_out[cnt] := status_to_ESR(s1, a1, DT_in, TX);
	X1 := S1;
	cnt := cnt + 1;
	esr_flag := TRUE;
END_IF;
IF s2 <> X2 AND ((s2 < 100) OR (S2 > 99 AND S2 < 200 AND mode >= 2) OR (S2 > 199 AND mode = 3)) THEN
	esr_out[cnt] := status_to_ESR(s2, a2, DT_in, TX);
	X2 := S2;
	cnt := cnt + 1;
	esr_flag := TRUE;
END_IF;
IF s3 <> X3 AND ((s3 < 100) OR (S3 > 99 AND S3 < 200 AND mode >= 2) OR (S3 > 199 AND mode = 3)) THEN
	esr_out[cnt] := status_to_ESR(s3, a3, DT_in, TX);
	X3 := S3;
	cnt := cnt + 1;
	esr_flag := TRUE;
END_IF;
IF cnt < 4 AND s4 <> X4 AND ((s4 < 100) OR (S4 > 99 AND S4 < 200 AND mode >= 2) OR (S4 > 199 AND mode = 3)) THEN
	esr_out[cnt] := status_to_ESR(s4, a4, DT_in, TX);
	X4 := S4;
	cnt := cnt + 1;
	esr_flag := TRUE;
END_IF;
IF cnt < 4 AND s5 <> X5 AND ((s5 < 100) OR (S5 > 99 AND S5 < 200 AND mode >= 2) OR (S5 > 199 AND mode = 3)) THEN
	esr_out[cnt] := status_to_ESR(s5, a5, DT_in, TX);
	X5 := S5;
	cnt := cnt + 1;
	esr_flag := TRUE;
END_IF;
IF cnt < 4 AND s6 <> X6 AND ((s6 < 100) OR (S6 > 99 AND S6 < 200 AND mode >= 2) OR (S6 > 199 AND mode = 3)) THEN
	esr_out[cnt] := status_to_ESR(s6, a6, DT_in, TX);
	X6 := S6;
	cnt := cnt + 1;
	esr_flag := TRUE;
END_IF;
IF cnt < 4 AND s7 <> X7 AND ((s7 < 100) OR (S7 > 99 AND S7 < 200 AND mode >= 2) OR (S7 > 199 AND mode = 3)) THEN
	esr_out[cnt] := status_to_ESR(s7, a7, DT_in, TX);
	X7 := S7;
	cnt := cnt + 1;
	esr_flag := TRUE;
END_IF;


(* revision history
hm	26. jan 2007		rev 1.0
	original version

hm	17. sep 2007	rev 1.1
	replaced time() with T_PLC_MS() for compatibility reasons
	
*)
END_FUNCTION_BLOCK

(* POU Other/status_to_ESR, ST *)
FUNCTION status_to_ESR : esr_data
VAR_INPUT
	status : BYTE;
	adress : STRING(10);
	DT_in : DT;
	TS : TIME;
END_VAR
VAR
END_VAR

(*
version 1.0	6 oct 2006
programmer 	hugo
tested by		tobias

status_to_esr creates esr data from a status byte.

*)
IF status < 100 THEN
	status_to_ESR.typ := 1;
ELSIF status < 200 THEN
	status_to_ESR.typ := 2;
ELSE
	status_to_ESR.typ := 3;
END_IF;
status_to_ESR.adress:= adress;
status_to_ESR.DS := DT_in;
status_to_ESR.TS := TS;
status_to_ESR.data[0] := status;
END_FUNCTION

(* POU XTEST/Baustein Tests/gen_rdt_test, CFC *)
PROGRAM gen_rdt_test
VAR
	x1: GEN_RDT;
	out: BOOL;
	start: BOOL;
	x2: TP;
	o2: BOOL;
END_VAR
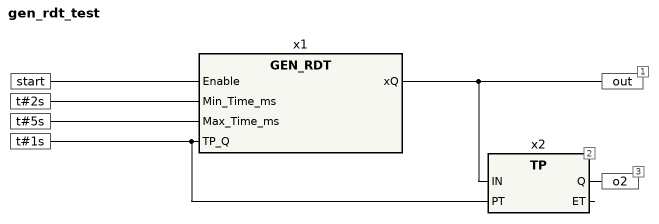
_CFC_ (* Continuous Function Chart, elements in execution order *)
#0 x1:GEN_RDT(Enable: start, Min_Time_ms: t#2s, Max_Time_ms: t#5s, TP_Q: t#1s)
#1 out <= #0.xQ
#2 x2:TP(IN: #0.xQ, PT: t#1s)
#3 o2 <= #2.Q
_END_CFC_
(* the same logic as Structured Text *)
x1(Enable := start, Min_Time_ms := t#2s, Max_Time_ms := t#5s, TP_Q := t#1s);
out := x1.xQ;
x2(IN := x1.xQ, PT := t#1s);
o2 := x2.Q;
END_PROGRAM

(* POU Engineering/signal generators/GEN_RDT, ST *)
FUNCTION_BLOCK GEN_RDT

VAR_INPUT
		 Enable		 	: BOOL := TRUE ;
		 Min_Time_ms	: TIME := t#1s ; (* min Taktzeit *)
		 Max_Time_ms	: TIME := t#1.2s ; (* Max Taktzeit *)
		 TP_Q		 		: TIME := t#100ms ; (* Zeit Ausgang auf TRUE *)
END_VAR
VAR_OUTPUT
		 xQ		 : BOOL ;
END_VAR
VAR
(* Taktgenerator Simulation *)
		 tonRDMTimer		: TON ; (* Zeitbaustein Taktgenerator *)
		 tof_xQ		 		: TOF ; (* Ausschaltverzögerung Taktgenerator *)
		 tRDMTime		: TIME ; (* Sollzeit *)
		 rRDMTime		: REAL ; (* Zufalswert Timer *)
END_VAR

(*
version 1.2	1 nov 2007
programmer 	J. Schohaus
tested by		Hugo

RDMT generates a defined pulse with pulse width TP_Q at random times. the random time will be defined with an minimum and maximum time.

*)


(*
FUNCTION_BLOCK RDMTimer
###############################################################################
		 Ersteller / author :		 		 		 		 		 J.Schohaus
		 Datum / date:		 		 		 		 		 		 13.07.2007
###############################################################################
		 Änderungen / Datum / Ersteller :		 		 		 		 		 		 		 		 		 		 		 		 		 		 		 
		 moditication / date / author :		 		 
###############################################################################
		 Verwendete Bibliotheken		 ( * werden im Baustein nicht benötigt )
		 		 		 		 Oscat.lib
###############################################################################
Beschreibung:
*)
tonRDMTimer ( IN:= Enable , PT:= tRDMTime );
tof_xQ ( IN:= tonRDMTimer.Q , PT:= TP_Q );
XQ := tof_xq.Q;
IF tonRDMTimer.Q THEN
		 xQ := TRUE ;
		 rRDMTime := RDM ( last:= rRDMTime ) ;
		 tRDMTime := REAL_TO_TIME ( rRDMTime * TIME_TO_DINT( Max_Time_ms - Min_Time_ms ) + TIME_TO_DINT(Min_Time_ms )) ;
		 tonRDMTimer ( IN:= FALSE );
END_IF;

(* revision history
J. Schohaus	19. nov 2007		rev 1.0
	origial version

*)
END_FUNCTION_BLOCK

(* POU XTEST/Baustein Tests/heat_meter_test, CFC *)
PROGRAM heat_meter_test
VAR
	kj : REAL;
	x1: heat_meter;
	run: BOOL;
	rst: BOOL;
	den: REAL;
	ent: REAL;
	x2: TP;
	clk: BOOL;
	kj1: REAL;
	x3: heat_meter;
END_VAR
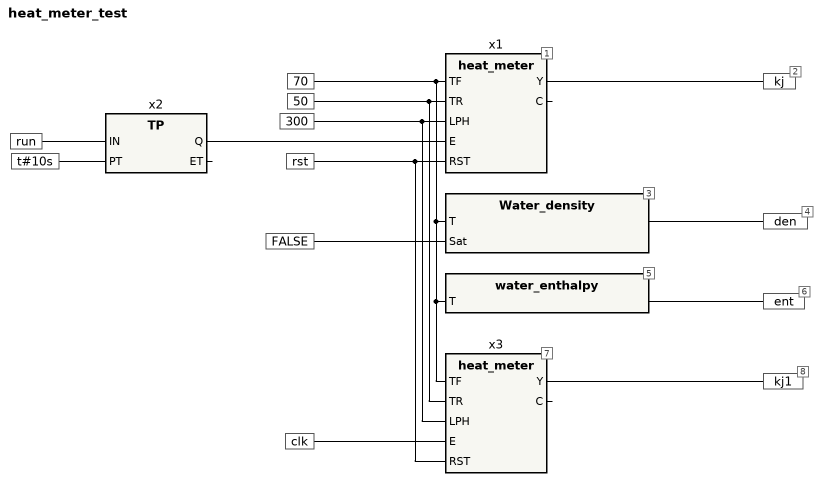
_CFC_ (* Continuous Function Chart, elements in execution order *)
#0 x2:TP(IN: run, PT: t#10s)
#1 x1:heat_meter(TF: 70, TR: 50, LPH: 300, E: #0.Q, RST: rst)
#2 kj <= #1.Y
#3 Water_density(T: 70, Sat: FALSE)
#4 den <= #3
#5 water_enthalpy(T: 70)
#6 ent <= #5
#7 x3:heat_meter(TF: 70, TR: 50, LPH: 300, E: clk, RST: rst, Pulse_Mode := TRUE)
#8 kj1 <= #7.Y
_END_CFC_
END_PROGRAM

(* POU Building/HLK/heat_meter, ST *)
FUNCTION_BLOCK heat_meter
VAR_INPUT
	TF, TR : REAL;
	LPH : REAL;
	E : BOOL;
	RST : BOOL;
END_VAR
VAR_INPUT CONSTANT
	CP : REAL;
	Density : REAL;
	Content : REAL;
	Pulse_Mode : BOOL;
	Return_meter : BOOL;
	AVG_time : TIME := T#5s;
END_VAR
VAR_OUTPUT
	Y : REAL;
	C : REAL;
END_VAR
VAR
	tx, last : DWORD;
	int1 : FT_INT;
	edge : BOOL;
	X: REAL;
	init: BOOL;
	Y_last: REAL;
END_VAR

(*
version 1.2	6. mar 2008
programmer 	hugo
tested by		tobias

Heat meter measures the heat transfer of water of a mixture of water and another component.
The inputs are foreward temperature and reverse temperature.
the additional component is specified with its parameters density, Specific heat capacity and content in %.
an input e anables the measurement while it can be configured to be based on X liters / pulse or in liters / hour.
the output is in Joule.

*)
IF rst THEN
	int1(rst := TRUE);
	int1.rst := FALSE;
	C := 0;
	Y := 0;
ELSIF pulse_mode AND e AND NOT edge THEN
	IF return_meter THEN
		X := (Water_density(TR, FALSE) * (water_enthalpy(TF) - water_enthalpy(TR)) * (1-content) + CP * Density * content*(TF-TR));
	ELSE
		X := (Water_density(TF, FALSE) * (water_enthalpy(TF) - water_enthalpy(TR)) * (1-content) + CP * Density * content*(TF-TR));
	END_IF;
	Y := Y + X * LPH;
ELSIF NOT pulse_mode AND e THEN
	IF return_meter THEN
		X := (Water_density(TR, FALSE) * (water_enthalpy(TF) - water_enthalpy(TR)) * (1-content) + CP * Density * content*(TF-TR));
	ELSE
		X := (Water_density(TF, FALSE) * (water_enthalpy(TF) - water_enthalpy(TR)) * (1-content) + CP * Density * content*(TF-TR));
	END_IF;
	int1(in := X * LPH / 3600.0, out_min := 0, out_max := 3E38);
	Y := int1.Out;
END_IF;

(* store the value of e *)
edge := e;

(* read system_time *)
tx := T_PLC_MS();

(* only init at startup necessary *)
IF NOT init THEN
	init := TRUE;
	last := tx;
END_IF;

(* calculate the current consumption *)
IF (tx - last >= TIME_TO_DWORD(AVG_TIME)) AND (avg_time > T#0s) THEN
	last := tx;
	C := (Y - Y_last) * 3.6/TIME_TO_DWORD(AVG_TIME);
	Y_last := Y;
END_IF;



(* revision history
hm		16.11.2007	rev 1.0
	original version

hm		24.12.2007	rev 1.1
	added config variable return_meter
	added output C for current consumption

hm		6. mar. 2008	rev 1.2
	corrected an error in pulse mode

*)
END_FUNCTION_BLOCK

(* POU Building/HLK/Water_density, ST *)
FUNCTION Water_density : REAL
VAR_INPUT
	T : REAL;
	Sat : BOOL;
END_VAR
VAR CONSTANT
	a0 : REAL := 999.83952;
	a1 : REAL := 16.952577;
	a2 : REAL := -7.9905127E-3;
	a3 : REAL := -4.6241757E-5;
	a4 : REAL := 1.0584601E-7;
	a5 : REAL := -2.8103006E-10;
	b  : REAL := 0.0168872;
END_VAR
VAR
	T2: REAL;
	T4: REAL;
END_VAR


(*
version 1.1	2 dec 2007
programmer 	hugo
tested by		tobias

this function calculates the water density for air free water between 0 and 100 deg C
while sat is false the denisty is calculated for air free water and when sat = true
the calculation is performed for water saturated with air.

*)
T2 := T * T;
T4 := T2 * T2;

(* original code changed for performance
Water_density := (a0 + a1*T + a2*EXPT(T,2) + a3*EXPT(t,3) + a4*EXPT(t,4) + a5*EXPT(t,5)) / (1 + b*T);
*)
Water_density := (a0 + a1*T + a2*T2 + a3*T2*T + a4*T4 + a5*T4*T) / (1 + b*T);

IF sat THEN Water_density := Water_density - 0.004612 + 0.000106 * T; END_IF;


(* revision history

hm	13.9.2007		rev 1.0
	original version

hm	2.12.2007		rev 1.1
	changed code for better performance
*)

(*
    °C - die Celsius-Temperatur in Grad Celsius
    v – das spezifische Volumen in Kubikdezimeter je Kilogramm dm³/kg
    h – die spezifische Enthalpie in Kilojoule je Kilogramm 	kJ/kg
    u – die spezifische Innere Energie in Kilojoule je Kilogramm 	kJ/kg
    s – die spezifische Entropie in Kilojoule je Kilogramm mal Kelvin 	kJ/(kg·K)
    cp - die spezifische Wärmekapazität bei konstantem Druck in Kilojoule je Kilogramm mal Kelvin 	kJ/(kg·K)
    Y – Volumenausdehnungskoeffizient in 10-3 durch Kelvin  10-3/K
    L – Wärmeleitfähigkeit in Milliwatt je Meter mal Kelvin  mW / (m·K) 
    n – Viskosität in Mikropascal mal Sekunde uPa·s 	
    s ? – Oberflächenspannung in Millinewton je Meter  mN/m


°C 		v 				h 			u 		s 			cp 		Y 		L		n		s	
-20		1,006580	
0 		1,000160 		0,06 		-0,04 	-0,0001 	4,228 	-0,080 	561,0 	1792 	75,65
4		1,000028
5 		1,0000 		21,1 		21,0 	0,076 		4,200 	0,011 	570,6 	1518 	74,95
10 		1,0003 		42,1 		42,0 	0,151 		4,188 	0,087 	580,0 	1306 	74,22
15 		1,0009 		63,0 		62,9 	0,224 		4,184 	0,152 	589,4 	1137 	73,49
20 		1,001797 		83,9 		83,8 	0,296 		4,183 	0,209 	598,4 	1001 	72,74
25 		1,0029 		104,8 		104,7 	0,367 		4,183 	0,259 	607,2 	890,4 	71,98
30 		1,0044 		125,8 		125,7 	0,437 		4,183 	0,305 	615,5 	797,7 	71,20
35 		1,0060 		146,7 		146,6 	0,505 		4,183 	0,347 	623,3 	719,6 	70,41
40 		1,007842 		167,58 	167,5 	0,572 		4,182 	0,386 	630,6 	653,3 	69,60
45 		1,0099 		188,5 		188,4 	0,638 		4,182 	0,423 	637,3 	596,3 	68,78
50 		1,0121 		209,4 		209,3 	0,704 		4,181 	0,457 	643,6 	547,1 	67,95
60 		1,017089 		251,2 		251,1 	0,831 		4,183 	0,522 	654,4 	466,6 	66,24
70 		1,0227 		293,1 		293,0 	0,955 		4,187 	0,583 	663,1 	404,1 	64,49
80 		1,029027 		335,0 		334,9 	1,075 		4,194 	0,640 	670,0 	354,5 	62,68
90 		1,0359 		377,0 		376,9 	1,193 		4,204 	0,696 	675,3 	314,6 	60,82
99,63 	1,0431 		417,5 		417,4 	1,303 		4,217 	0,748 	679,0 	283,0 	58,99
100	1,043453		419,1

Stoffdaten von Wasser Quelle Wickipedia

*)
END_FUNCTION

(* POU Building/HLK/water_enthalpy, ST *)
FUNCTION water_enthalpy : REAL
VAR_INPUT
	T : REAL;
END_VAR
VAR
	Pts : INT := 11;
	data : ARRAY[1..20, 0..1] OF REAL := 0,0.06, 10,42.1, 20,83.9, 30,125.8, 40,167.58, 50,209.4, 60,251.2, 70,293.1, 80,335.0, 90, 377.0, 100,419.1 ;
END_VAR

(*
version 1.0	29 oct 2007
programmer 	hugo
tested by		tobias

water_enthalpy calculates the enthalpy of liquid water from 0..100 °C 

*)
water_enthalpy := LINEAR_INT(T, Data, Pts);


(* revision history

hm	29.10.2007	rev 1.0
	original version

*)

(*
    °C - die Celsius-Temperatur in Grad Celsius
    v – das spezifische Volumen in Kubikdezimeter je Kilogramm dm³/kg
    h – die spezifische Enthalpie in Kilojoule je Kilogramm 	kJ/kg
    u – die spezifische Innere Energie in Kilojoule je Kilogramm 	kJ/kg
    s – die spezifische Entropie in Kilojoule je Kilogramm mal Kelvin 	kJ/(kg·K)
    cp - die spezifische Wärmekapazität bei konstantem Druck in Kilojoule je Kilogramm mal Kelvin 	kJ/(kg·K)
    Y – Volumenausdehnungskoeffizient in 10-3 durch Kelvin  10-3/K
    L – Wärmeleitfähigkeit in Milliwatt je Meter mal Kelvin  mW / (m·K) 
    n – Viskosität in Mikropascal mal Sekunde uPa·s 	
    s ? – Oberflächenspannung in Millinewton je Meter  mN/m


°C 		v 				h 			u 		s 			cp 		Y 		L		n		s	
-20		1,006580	
0 		1,000160 		0,06 		-0,04 	-0,0001 	4,228 	-0,080 	561,0 	1792 	75,65
4		1,000028
5 		1,0000 		21,1 		21,0 	0,076 		4,200 	0,011 	570,6 	1518 	74,95
10 		1,0003 		42,1 		42,0 	0,151 		4,188 	0,087 	580,0 	1306 	74,22
15 		1,0009 		63,0 		62,9 	0,224 		4,184 	0,152 	589,4 	1137 	73,49
20 		1,001797 		83,9 		83,8 	0,296 		4,183 	0,209 	598,4 	1001 	72,74
25 		1,0029 		104,8 		104,7 	0,367 		4,183 	0,259 	607,2 	890,4 	71,98
30 		1,0044 		125,8 		125,7 	0,437 		4,183 	0,305 	615,5 	797,7 	71,20
35 		1,0060 		146,7 		146,6 	0,505 		4,183 	0,347 	623,3 	719,6 	70,41
40 		1,007842 		167,58 	167,5 	0,572 		4,182 	0,386 	630,6 	653,3 	69,60
45 		1,0099 		188,5 		188,4 	0,638 		4,182 	0,423 	637,3 	596,3 	68,78
50 		1,0121 		209,4 		209,3 	0,704 		4,181 	0,457 	643,6 	547,1 	67,95
60 		1,017089 		251,2 		251,1 	0,831 		4,183 	0,522 	654,4 	466,6 	66,24
70 		1,0227 		293,1 		293,0 	0,955 		4,187 	0,583 	663,1 	404,1 	64,49
80 		1,029027 		335,0 		334,9 	1,075 		4,194 	0,640 	670,0 	354,5 	62,68
90 		1,0359 		377,0 		376,9 	1,193 		4,204 	0,696 	675,3 	314,6 	60,82
99,63 	1,0431 		417,5 		417,4 	1,303 		4,217 	0,748 	679,0 	283,0 	58,99
100	1,043453		419,1

Stoffdaten von Wasser Quelle Wickipedia

Wasser hat unter Normaldruck seine größte Dichte von 1000 Kilogramm pro Kubikmeter bei 3,98 °C und zeigt damit eine Dichteanomalie. 
Diese besteht darin, dass sich Wasser unterhalb von 3,98 °C bei weiterer Temperaturverringerung, auch beim Wechsel zum festen 
Aggregatzustand, wieder ausdehnt, was man nur von wenigen Stoffen kennt. Die derzeit genauesten publizierten Werte für die maximale 
Dichte liegen bei (999,974950 ± 0,00084) kg/m³ und bei (3,983 ± 0,00067) °C für die Temperatur, bei der dieser Wert erreicht wird. 
Die Werte stellen einen Mittelwert der von verschiedenen physikalischen Instituten veröffentlichten Zahlen dar (Stand 2001).

Die Berechnung der Dichte von luftfreiem Wasser DLF in Abhängigkeit von der Temperatur T ([T] = °C) kann mit Hilfe der folgenden 
Virialgleichung erfolgen:
: \frac{D_{\rm LF}}{\rm g/l} = \frac{a_0 + a_1 T + a_2 T^2 + a_3 T^3 + a_4 T^4 + a_5 T^5}{1 + b T}.
mit den Koeffizienten: a0 = 999,83952; a1 = 16,952577 (°C)-1; a2 = -7,9905127·10-3 (°C)-2; a3 = -4,6241757·10-5 (°C)-3; 
a4 = 1,0584601·10-7 (°C)-4; a5 = -2,8103006·10-10 (°C)-5 und b = 0,0168872. 
Für die Berechnung der Dichte von luftgesättigtem Wasser korrigiert man den Wert nach 
DLG/(g/l) = DLF/(g/l) - 0,004612 + 0,000106 (°C)-1·T. (Quelle: PTB-Mitteilungen 100/3-90)

*)
END_FUNCTION

(* POU Mathematical/functions/LINEAR_INT, ST *)
FUNCTION LINEAR_INT : REAL
VAR_INPUT
	X : REAL;
	XY : ARRAY[1..20,0..1] OF REAL;
	Pts : INT;
END_VAR
VAR
	i : INT;
END_VAR

(*
	version 1.1	27 dec 2007
	programmer 	oscat
	tested BY		oscat

LINEAR_INT calculates an output based on a linear interpolation of up to 20 coordinates given in an array
the input coordinates have to start at the lowest array position and must be sorted ba ascending X values.

*)
(*make sure n is bound within the array size *)
pts := MIN(pts,20);

(* calculate the linear segement interpolation *)
i := 2;
(* search for segment and calculate output
	below and above the defined segments we interpolate the last segment *)
WHILE (i < pts) AND (XY[i,0] < X) DO
	i := i + 1;
END_WHILE;

(* calculate the output value on the corresponding segment coordinates *)
LINEAR_INT := ((XY[i,1] - XY[i-1,1]) * X - XY[i,1] * XY[i-1,0] + XY[i-1,1] * XY[i,0]) / (XY[i,0] - XY[i-1,0]);

(* revision history
hm	7. oct 2007		rev 1.0
	original version

hm	27 dec 2007		rev 1.1
	changed code for better performance
*)
END_FUNCTION

(* POU XTEST/Baustein Tests/holiday_test, CFC *)
PROGRAM holiday_test
VAR
	x1: holiday;
	dtin: DATE;
	hol: BOOL;
	nameh: STRING;
END_VAR
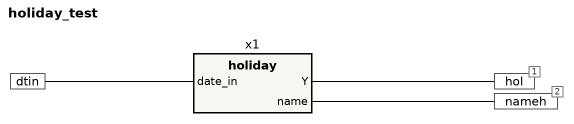
_CFC_ (* Continuous Function Chart, elements in execution order *)
#0 x1:holiday(date_in: dtin)
#1 hol <= #0.Y
#2 nameh <= #0.name
_END_CFC_
(* the same logic as Structured Text *)
x1(date_in := dtin);
hol := x1.Y;
nameh := x1.name;
END_PROGRAM

(* POU Time&Date/holiday, ST *)
FUNCTION_BLOCK holiday
VAR_INPUT
	date_in : DATE;
END_VAR
VAR_INPUT CONSTANT
	size : INT := 24;
	feiertag : ARRAY [0..24] OF STRING(27) := 'Neujahr', 'Heilig Drei Könige', 'Karfreitag', 'Ostersonntag', 'Ostermontag', 'Tag der Arbeit',
	'Christi Himmelfahrt', 'Pfingstsonntag', 'Pfingstmontag', 'Fronleichnam', 'Augsburger Friedensfest', 'Maria Himmelfahrt',
	'Tag der Deutschen Einheit', 'Reformationstag', 'Allerheiligen', 'Buss und Bettag', '1. Weihnachtstag', '2. Weihnachtstag';
	f_day : ARRAY [0..24] OF SINT := 1, 6, -2, 0, 1, 1, 39, 49, 50 , 60, 8, 15, 3, 31, 1, 23, 25, 26;
	f_month : ARRAY [0..24] OF SINT := 1, 1, 0, 0, 0, 5, 0, 0, 0, 0, 8, 8, 10, 10, 11, 11, 12, 12;
	(* if month = 0 then F_day is the offset in days from easter *)
	f_use : ARRAY [0..24] OF SINT := 1,1,1,1,1,1,1,1,1,1,0,1,1,0,1,0,1,1;
	(* 0 = not used, 1 = used, -1..-7 menas the weekday before the specified date example -3 means wednesday before 23.11 *)
	Friday : BOOL := FALSE;
	Saturday : BOOL := FALSE;
	Sunday : BOOL := FALSE;
END_VAR
VAR_OUTPUT
	Y : BOOL;
	name : STRING(20);
END_VAR
VAR
	last_active : DATE;
	ostern: DATE;
	i: INT;
	jahr: INT;
	x_date: DATE;
	wday : INT;
END_VAR

(*
version 1.3	24 nov 2007
programmer 	hugo
tested by		tobias

holiday calculates if a given day is a holiday and displays the name of the holiday as string as well as a boolean flag to indicate a holiday.
the holidays can be specified in an array in the constants section of the function block.
a holiday can be of fixed date for example new years day on january 1st.
a holiday can have a fixed offset from easter sunday as for most church holidays.
a holiday can be a specific weekday before a fixed date, for example buss und bettag is the last wednesday before nov 23rd.
with a simple f_use flag any specific holiday can be turned on or off if needed.
The setup Variables Friday, Saturday and Sunday can be used to activate the output on the specific weekday.

*)
(* for performance reasons only activate once a day *)
IF last_active = date_in THEN RETURN; END_IF;

(* berechnung von ostern für das aktuelle jahr *)
jahr := year(date_in);
Ostern := easter(jahr);
last_active := Date_in;

(* check array if today is holiday *)
Y := FALSE;
name := '';
FOR i := 0 TO size DO
	x_date := set_Date(jahr, f_month[i], f_day[i]);
	IF f_use[i] = 1 AND f_month[i] > 0 THEN
		(* check for fixed date holiday *)
		IF x_date = date_in THEN
			Y := TRUE;
			name := feiertag[i];
			RETURN;
		END_IF;
	ELSIF f_use[i] = 1 AND f_month[i] = 0 THEN
		(* check for holiday in reference to easter *)
		IF date_add(ostern,f_day[i] ,0,0,0) = date_in THEN
			Y := TRUE;
			name := feiertag[i];
			RETURN;
		END_IF;
	ELSIF f_use[i] < 0 THEN
		(* check for holiday on a weekday before date *)
		IF weekday(date_in) = ABS(f_use[i]) AND date_in < x_date AND date_in >= date_add(x_date,-7,0,0,0) THEN
			Y := TRUE;
			name := feiertag[i];
			RETURN;
		END_IF;
	END_IF;
END_FOR;

wday := weekday(date_in);
IF wday = 7 AND Sunday THEN
	Y := TRUE;
ELSIF wday = 6 AND Saturday THEN
	Y := TRUE;
ELSIF wday = 5 AND Friday THEN
	Y := TRUE;
END_IF;

(* revision history
hm 27.2.2007		rev 1.1
	deleted unused variable init

hm	31 oct 2007	rev 1.2
	changed holiday definition from constant to input constant to allow easier changes by user without recompilation of the lib

hm 24 nov 2007	rev 1.3
	changes F_use of  Buß_und_Bettag to 0 because this is no official holiday
*)

(*
Neujahrstag 	1. Januar 	• 	• 	• 	• 	• 	• 	• 	• 	• 	• 	• 	• 	• 	• 	• 	•
Heilige Drei Könige 	6. Januar 	• 	• 												• 		
Karfreitag 	Ostersonntag - 2d 	• 	• 	• 	• 	• 	• 	• 	• 	• 	• 	• 	• 	• 	• 	• 	•
Ostersonntag 	siehe Osterdatum 				(•) 												
Ostermontag 	Ostersonntag + 1d 	• 	• 	• 	• 	• 	• 	• 	• 	• 	• 	• 	• 	• 	• 	• 	•
Tag der Arbeit 	1. Mai 	• 	• 	• 	• 	• 	• 	• 	• 	• 	• 	• 	• 	• 	• 	• 	•
Christi Himmelfahrt 	Ostersonntag + 39d 	• 	• 	• 	• 	• 	• 	• 	• 	• 	• 	• 	• 	• 	• 	• 	•
Pfingstsonntag 	Ostersonntag + 49d 				(•) 												
Pfingstmontag 	Ostersonntag + 50d 	• 	• 	• 	• 	• 	• 	• 	• 	• 	• 	• 	• 	• 	• 	• 	•
Fronleichnam 	Ostersonntag + 60d 	• 	• 					• 			• 	• 	• 	1) 			2)
Augsburger Friedensfest 	8. August 		(3) 														
Mariä Himmelfahrt 	15. August 		(5) 										• 				
Tag der Deutschen Einheit 	3. Oktober 6) 	• 	• 	• 	• 	• 	• 	• 	• 	• 	• 	• 	• 	• 	• 	• 	•
Reformationstag 	31. Oktober 				• 				• 					• 	• 		•
Allerheiligen 	1. November 	• 	• 								• 	• 	• 				
Buß- und Bettag 4) 	Mittwoch vor dem 23.11. 			7 										• 			
1. Weihnachtstag 	25. Dezember 	• 	• 	• 	• 	• 	• 	• 	• 	• 	• 	• 	• 	• 	• 	• 	•
2. Weihnachtstag 	26. Dezember 	• 	• 	• 	• 	• 	• 	• 	• 	• 	• 	• 	• 	• 	• 	• 	•
*)
END_FUNCTION_BLOCK

(* POU Time&Date/easter, ST *)
FUNCTION easter : DATE
VAR_INPUT
	year : INT;
END_VAR
VAR
	b,c: INT;
	oday: INT;
	omon: INT;
END_VAR

(*
version 1.2	3. feb 2008
programmer 	hugo
tested by		tobias

easter calculates the day of easter sunday for a given year.
most other catholic holidays are calculated in reference to easter sunday.

*)
(* this algorithms is 60 us *)

b := (204 - 11 * (year MOD 19)) MOD 30;
IF b > 27 THEN b := b - 1; END_IF;
c := (year + SHR(year,2) + b - 13) MOD 7;
oday := 28 + b - c;
IF oday > 33 THEN
    oday := oday - 31;
    omon := 4;
ELSE
	omon := 3;
END_IF;
easter := set_Date(year, omon, oday);



(* alternativer algorithmus ueber das pasah fest
execution time roughly 200us
Der sog. Passah-Vollmond wird berechnet, in dem das Jahr durch 19 ge-
teilt wird und der Rest mit der folgenden Tabelle verglichen wird:
 
    0: Apr 14       5: Apr 18      10: Mrz 25      15: Mrz 30
    1: Apr 03       6: Apr 08      11: Apr 13      16: Apr 17
    2: Mrz 23       7: Mrz 28      12: Apr 02      17: Apr 07
    3: Apr 11       8: Apr 16      13: Mrz 22      18: Mrz 27
    4: Mrz 31       9: Apr 05      14: Apr 10
 
Faellt dieses Datum auf einen Sonntag, ist Ostern der naechste Sonntag!
 
Beispiel: 1992 MOD 19 = 16, daraus folgt 17.04., der naechste Sonntag
          ist dann der 19. April (Ostersonntag)
*)


(* this algorithm is 180 us
a := year MOD 19;
b := year / 100;
c := year MOD 100;
d := b / 4;
e := b MOD 4;
f := (b + 8) / 25;
g := (b - f + 1) / 3;
h := (19 * a + b - d -g + 15) MOD 30;
i := C / 4;
k := c MOD 4;
l := (32 + 2*e + 2*i - h - k) MOD 7;
m := (a + 11 * h + 22 * l) / 451;
x := h + l - 7 * m + 114;
n := X / 31;
o := x MOD 31 + 1;

easter := set_Date(year,n,o);
*)
(*
Im Magazin "Nature" vom 20. April 1876 veröffentlichte ein anonymer Autor eine Tabelle mit Regeln zur Berechnung des (Gregorianischen) Ostersonntages des Jahres J. In Formeln ausgedrückt erhält man das Folgende:
a	=	J mod 19
b	=	int(J / 100)
c	=	J mod 100
d	=	int(b / 4)
e	=	b mod 4
f	=	int((b + 8) / 25)
g	=	int((b - f + 1) / 3
h	=	(19 · a + b - d - g + 15) mod 30
i	=	int(c / 4)
k	=	c mod 4
l	=	(32 + 2 · e + 2 · i - h - k) mod 7
m	=	int((a + 11 · h + 22 · l) / 451)
n	=	int((h + l - 7 · m + 114) / 31)
o	=	(h + l - 7 · m + 114) mod 31

n ist hierbei die Nummer des Monats, o + 1 die Nummer des Tages auf welchen der Ostersonntag im Jahr J fällt. Dieser Algorithmus kommt ohne Hilfszahlen aus.

*)

(* revision history
hm	27. dec 2006	rev 1.0
	original version

hm	15. dec 2007	rev 1.1
	modified code for better performance

hm	3. feb 2008		rev 1.2
	modified code for better performance
*)
END_FUNCTION

(* POU Time&Date/set_Date, ST *)
FUNCTION set_Date : DATE
VAR_INPUT
	year : INT;
	month : INT;
	day : INT;
END_VAR
VAR
	count : DWORD;
END_VAR

(*
version 1.2	3 jan 2008
programmer 	hugo
tested by		tobias

creates a date output from year, month and day of month   

*)
IF STEP7 THEN
	count := SHR(INT_TO_DWORD(year) * 1461 - 2907393,2)+day;
ELSE
	count := SHR(INT_TO_DWORD(year) * 1461 - 2878173,2)+day;
END_IF;

IF month < 5 THEN
	IF month < 3 THEN
		IF month = 2 THEN count := count + 31; END_IF;
	ELSE
		IF month = 4 THEN
			IF SHL(year,14) = 0 THEN count := count + 91; ELSE count := count + 90; END_IF;
		ELSE (* month = 3 *)
			IF SHL(year,14) = 0 THEN count := count + 60; ELSE count := count + 59; END_IF;
		END_IF;
	END_IF;
ELSIF month < 9 THEN
	IF month < 7 THEN
		IF month = 6 THEN
			IF SHL(year,14) = 0 THEN count := count + 152; ELSE count := count + 151; END_IF;
		ELSE (* month = 5 *)
			IF SHL(year,14) = 0 THEN count := count + 121; ELSE count := count + 120; END_IF;
		END_IF;
	ELSE
		IF month = 8 THEN
			IF SHL(year,14) = 0 THEN count := count + 213; ELSE count := count + 212; END_IF;
		ELSE (* month = 7 *)
			IF SHL(year,14) = 0 THEN count := count + 182; ELSE count := count + 181; END_IF;
		END_IF;
	END_IF;
ELSE (* month is 9 or higher *)
	IF month < 11 THEN
		IF month = 10 THEN
			IF SHL(year,14) = 0 THEN count := count + 274; ELSE count := count + 273; END_IF;
		ELSE (* month = 9 *)
			IF SHL(year,14) = 0 THEN count := count + 244; ELSE count := count + 243; END_IF;
		END_IF;
	ELSE
		IF month = 12 THEN
			IF SHL(year,14) = 0 THEN count := count + 335; ELSE count := count + 334; END_IF;
		ELSE (* month = 11 *)
			IF SHL(year,14) = 0 THEN count := count + 305; ELSE count := count + 304; END_IF;
		END_IF;
	END_IF;
END_IF;
set_Date := DWORD_TO_DATE(count * 86400);

(*  code before rev 1.4
leap := leap_year(year);
IF STEP7 THEN
	count := SHR((year-1)*1461-2905932+day*4,2);
ELSE
	count := SHR((year-1)*1461-2876712+day*4,2);
END_IF;
CASE month OF
2:	count := count + 31;
3:	IF leap THEN count := count + 60; ELSE count := count + 59; END_IF;
4:	IF leap THEN count := count + 91; ELSE count := count + 90; END_IF;
5:	IF leap THEN count := count + 121; ELSE count := count + 120; END_IF;
6:	IF leap THEN count := count + 152; ELSE count := count + 151; END_IF;
7:	IF leap THEN count := count + 182; ELSE count := count + 181; END_IF;
8:	IF leap THEN count := count + 213; ELSE count := count + 212; END_IF;
9:	IF leap THEN count := count + 244; ELSE count := count + 243; END_IF;
10:	IF leap THEN count := count + 274; ELSE count := count + 273; END_IF;
11:	IF leap THEN count := count + 305; ELSE count := count + 304; END_IF;
12:	IF leap THEN count := count + 335; ELSE count := count + 334; END_IF;
END_CASE;
set_Date := DWORD_TO_DATE(count * 86400);
*)

(* old code before rev 1.3
leap := leap_year(year);
IF STEP7 THEN
	count := TRUNC((year-1)*365.25-726483+day);
ELSE
	count := TRUNC((year-1)*365.25-719178+day);
END_IF;
CASE month OF
2:	count := count + 31;
3:	IF leap THEN count := count + 60; ELSE count := count + 59; END_IF;
4:	IF leap THEN count := count + 91; ELSE count := count + 90; END_IF;
5:	IF leap THEN count := count + 121; ELSE count := count + 120; END_IF;
6:	IF leap THEN count := count + 152; ELSE count := count + 151; END_IF;
7:	IF leap THEN count := count + 182; ELSE count := count + 181; END_IF;
8:	IF leap THEN count := count + 213; ELSE count := count + 212; END_IF;
9:	IF leap THEN count := count + 244; ELSE count := count + 243; END_IF;
10:	IF leap THEN count := count + 274; ELSE count := count + 273; END_IF;
11:	IF leap THEN count := count + 305; ELSE count := count + 304; END_IF;
12:	IF leap THEN count := count + 335; ELSE count := count + 334; END_IF;
END_CASE;
set_Date := DWORD_TO_DATE(count * 86400);
*)




(* revision history
hm	4. aug. 2006	rev 1.0
	original version

hm	19 sep. 2007	rev 1.1
	use function leap_year to calculate leap year, more exceptions are handled

hm	1. okt	2007	rev 1.2
	added compatibility to step7

hm	16.dec 2007		rev 1.3
	changed code to improove performance

hm	3. jan. 2008		rev 1.4
	further improvements in performance
*)
END_FUNCTION

(* POU Time&Date/month, ST *)
FUNCTION month : INT
VAR_INPUT
	idate : DATE;
END_VAR
VAR
END_VAR

(*
version 1.1	1 okt 2007
programmer 	hugo
tested by		tobias

returns the month of a year

*)
month := day_of_year(idate);
IF leap_of_Date(idate) THEN
	CASE month OF
		1..31 	:	month := 1;
		32..60	:	month := 2;
		61..91	:	month := 3;
		92..121 :	month := 4;
		122..152:	month := 5;
		153..182:	month := 6;
		183..213:	month := 7;
		214..244:	month := 8;
		245..274:	month := 9;
		275..305:	month := 10;
		306..335:	month := 11;
		336..366:	month := 12;
	END_CASE;
ELSE
	CASE month OF
		1..31 	:	month := 1;
		32..59	:	month := 2;
		60..90	:	month := 3;
		91..120 :	month := 4;
		121..151:	month := 5;
		152..181:	month := 6;
		182..212:	month := 7;
		213..243:	month := 8;
		244..273:	month := 9;
		274..304:	month := 10;
		305..334:	month := 11;
		335..365:	month := 12;
	END_CASE;
END_IF;


(* old code used in rev 1.0
month := STRING_TO_INT(MID(DATE_TO_STRING(idate),2,8));
*)

(* revision history
hm	1. aug 2006		rev 1.0
	original version	

hm	1. okt 2007		rev 1.1
	replaced old code (string conversion) with mathematics
	the execution time is now multiple times faster.

*)
END_FUNCTION

(* POU Time&Date/leap_of_Date, ST *)
FUNCTION leap_of_Date : BOOL
VAR_INPUT
	idate : DATE;
END_VAR
VAR
END_VAR

(*
version 1.2	8 jan 2008
programmer 	hugo
tested by		tobias

leap_year is true if the tested year is a leap year  

*)
leap_of_Date := SHL(DWORD_TO_INT((DATE_TO_DWORD(idate)+43200) / 31557600)+2,14) = 0;


(* change history

2.10.2006		rev 1.1
the function now calls leap_year to accomodate further accuracy.
the function now works for any year from 1970 to 2100

8. jan 2008		rev 1.2
	improved code for better performance
*)
END_FUNCTION

(* POU Time&Date/date_add, ST *)
FUNCTION date_add : DATE
VAR_INPUT
	idate : DATE;
	D : INT;
	W : INT;
	M : INT;
	Y : INT;
END_VAR
VAR
	mo: INT;
	yr : INT;
END_VAR


(*
version 1.2	1 nov 2007
programmer 	hugo
tested by		tobias

date_add adds days, weeks, month or years to a date.
negative inputs are allowed for subtraction.

*)
date_add := DWORD_TO_DATE(DATE_TO_DWORD(idate) + 86400 * INT_TO_DWORD(d) + 604800 * INT_TO_DWORD(w));
yr := year(date_add) + y;
IF m > 0 THEN
	mo := month(date_add) + m;
	yr := yr + (mo - 1) / 12;
	mo := mo MOD 12;
	IF mo = 0 THEN mo := 12; END_IF;
	date_add := set_Date(yr, mo, day_of_month(date_add));
ELSIF m < 0 THEN
	mo := month(date_add) + m;
	yr := yr + mo / 12 - 1;
	mo := mo MOD 12 + 12;
	date_add := set_Date(yr, mo, day_of_month(date_add));
ELSE
	date_add := set_Date(yr, month(date_add), day_of_month(date_add));
END_IF;

(* revision history

hm 27.12.2006	rev 1.0

hm 12.4.2007		rev 1.1
	corrected an error while date would be incorrect when year  = 0

hm	1.11.2007		rev 1.2
	added int_to_dword stetements to avoid possible overrun with möller ecp4
*)
END_FUNCTION

(* POU Time&Date/day_of_month, ST *)
FUNCTION day_of_month : INT
VAR_INPUT
	idate : DATE;
END_VAR
VAR
END_VAR

(*
version 1.4	8. jan 2008
programmer 	hugo
tested by		tobias

returns the day OF month for any DATE

*)
day_of_month := day_of_year(idate);
IF leap_of_Date(idate) THEN
	CASE day_of_month OF
		32..60	:	day_of_month := day_of_month - 31;
		61..91	:	day_of_month := day_of_month - 60;
		92..121 :	day_of_month := day_of_month - 91;
		122..152:	day_of_month := day_of_month - 121;
		153..182:	day_of_month := day_of_month - 152;
		183..213:	day_of_month := day_of_month - 182;
		214..244:	day_of_month := day_of_month - 213;
		245..274:	day_of_month := day_of_month - 244;
		275..305:	day_of_month := day_of_month - 274;
		306..335:	day_of_month := day_of_month - 305;
		336..366:	day_of_month := day_of_month - 335;
	END_CASE;
ELSE
	CASE day_of_month OF
		32..59	:	day_of_month := day_of_month - 31;
		60..90	:	day_of_month := day_of_month - 59;
		91..120 :	day_of_month := day_of_month - 90;
		121..151:	day_of_month := day_of_month - 120;
		152..181:	day_of_month := day_of_month - 151;
		182..212:	day_of_month := day_of_month - 181;
		213..243:	day_of_month := day_of_month - 212;
		244..273:	day_of_month := day_of_month - 243;
		274..304:	day_of_month := day_of_month - 273;
		305..334:	day_of_month := day_of_month - 304;
		335..365:	day_of_month := day_of_month - 334;
	END_CASE;
END_IF;


(*
this function is simple but took too long with 133 us
the problem is date_to_string is far too slow
day_of_month := STRING_TO_INT(RIGHT(DATE_TO_STRING(idate),2));

Revision history

hm 22.1.2007		rev 1.1
	deleted unused variable day_in_year and day_in_year_begin

hm	1. okt 2007		rev 1.2
	changed code to use day_of_year and leap_of_date
	added compatibility to STEP7

hm	8. oct 2007		rev 1.3
	deleted unused variable yr

hm	8. jan 2008		rev 1.4
	improved performance
*)
END_FUNCTION

(* POU Time&Date/weekday, ST *)
FUNCTION weekday : INT
VAR_INPUT
	idate : DATE;
END_VAR
VAR
END_VAR

(*
version 1.2	23 dec 2007
programmer 	hugo
tested by		tobias

calculates the weekday of a week according to ISO8601   
monday = 1 ..... sunday = 7  

*)
IF step7 THEN
	weekday := DWORD_TO_INT((DATE_TO_DWORD(idate)/86400+6) MOD 7) + 1;
ELSE
	weekday := DWORD_TO_INT((DATE_TO_DWORD(idate)/86400+3) MOD 7) + 1;
END_IF;
(* revision history
hm 21.8.06 rev 1.1
	corrected a miscalculation

hm	23.12.2007	rev 1.2
	correction for step7

*)
END_FUNCTION

(* POU XTEST/Baustein Tests/interpol_test, CFC *)
PROGRAM interpol_test
VAR
	wd: REAL;
	sat: BOOL;
	x3: FT_rmp;
	in: REAL;
	ilin: REAL;
	ARR: ARRAY [1..20,0..1] OF REAL :=  -10,-0.53, 10,0.53, 100,88.3, 200,122.2;
	ARRp: ARRAY [1..5,0..1] OF REAL :=  -10,-0.53, 10,0.53, 100,88.3, 200,122.2;
	ipol: REAL;
END_VAR
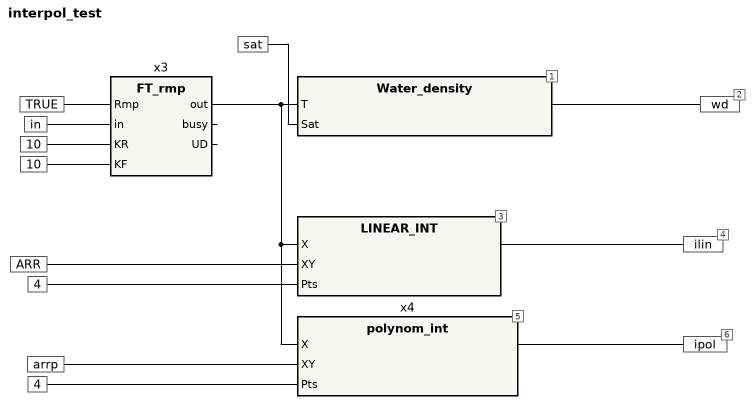
_CFC_ (* Continuous Function Chart, elements in execution order *)
#0 x3:FT_rmp(Rmp: TRUE, in: in, KR: 10, KF: 10)
#1 Water_density(T: #0.out, Sat: sat)
#2 wd <= #1
#3 LINEAR_INT(X: #0.out, XY: ARR, Pts: 4)
#4 ilin <= #3
#5 x4:polynom_int(X: #0.out, XY: arrp, Pts: 4)
#6 ipol <= #5
_END_CFC_
END_PROGRAM

(* POU Mathematical/functions/FT_rmp, ST *)
FUNCTION_BLOCK FT_rmp
VAR_INPUT
	Rmp : BOOL := TRUE;
	in : REAL;
	KR : REAL;
	KF : REAL;
END_VAR
VAR_OUTPUT
	out : REAL;
	busy : BOOL;
	UD : BOOL;
END_VAR
VAR
	tx: TIME;
	last: TIME;
	init: BOOL;
END_VAR

(*
	version 1.4	25 jan 2008
	programmer 	oscat
	tested BY		oscat

this ramp function follows an input signal with a linear ramp up or down, the up or down speed can be set with KF and KR.
a K factor of 1 means 1 unit per second on the output. K factors can only be positive and not negative.
a busy output signals the ramp is running or busy false means the in value is present on the output.
a rmp input false means the output follows the input dierctly while a rmp = true means the output follows the input with a ramp.
a updn output signal the directon of the ramp (up or down).

*)
(* read system time *)
tx := DWORD_TO_TIME(T_PLC_MS()) - last;

IF NOT init THEN
	init := TRUE;
	last := tx;
	tx := t#0s;
	out := in;
END_IF;
IF NOT rmp THEN
	out := in;
	busy := FALSE;
ELSIF out > in THEN
	(* ramp down *)
	out := out - TIME_TO_REAL(tx) * 0.001 * KF;
	out := MAX(in, out);
ELSIF out < in THEN
	(* ramp up *)
	out := out + TIME_TO_REAL(tx) * 0.001 * KR;
	out := MIN(in, out);
END_IF;

(* set busy and dir flags *)
IF out < in THEN
	busy := TRUE;
	ud := 1;
ELSIF out > in THEN
	busy := TRUE;
	ud := 0;
ELSE
	busy := FALSE;
END_IF;
last := last + tx;


(* revision history:

hm 8.10.2006			rev 1.1
	added ud output

hm 12. feb 2007		rev 1.2
	added init variable and corrected a possible startup problem

hm	17. sep 2007	rev 1.3
	replaced time() with t_plc_ms() for compatibility reasons

hm	25. jan 2008	rev 1.4
	performance improvements
	allow KR and KF to be 0
*)
END_FUNCTION_BLOCK

(* POU Mathematical/functions/POLYNOM_INT, ST *)
FUNCTION POLYNOM_INT : REAL
VAR_INPUT
	X : REAL;
	XY : ARRAY[1..5,0..1] OF REAL;
	Pts : INT;
END_VAR
VAR
	I, J : INT;
	stop: INT;
END_VAR

(*
	version 1.2	22 feb 2008
	programmer 	oscat
	tested BY		oscat

POLYNOM_INT calculates an output based on a Polynom interpolation of up to 5 coordinates given in an array
the indut coordinates have to start at the lowest array position and must be sorted ba ascending X values.

*)
(*make sure n is bound within the array size *)
pts := MIN(pts, 5);

(* this part is only to calculate the polynom parameters, which are then stores in the Y array
	the array values, it is not needed during runtime, unless the parameters will change during runtime
	the remaining code without this setup code can be used within a function to calculate specific functions
	the content of the arrays is then used as constant values within the function *)

FOR i := 1 TO pts DO
	stop := i + 1;
   	FOR j := pts TO stop BY -1 DO
   		XY[j,1] := (XY[j,1] - XY[j-1,1]) / (XY[j,0] - XY[j-i,0]);
	END_FOR;
END_FOR;


(* this part is the actual calculation *)
POLYNOM_INT := 0;
FOR i := pts TO 1 BY -1 DO
       POLYNOM_INT := POLYNOM_INT * (X - XY[i,0]) + XY[i,1];
END_FOR;


(* revision history
hm		8. okt 2007		rev 1.0
	original version

hm		17. dec 2007	rev 1.1
	init makes no sense for a function

hm		22. feb 2008	rev 1.2
	improved performance
*)
END_FUNCTION

(* POU XTEST/Baustein Tests/meter_test, CFC *)
PROGRAM meter_test
VAR
	x1: Meter;
	x2: METER_STAT;
	m1, m2: REAL;
	I1, I2:BOOL;
	divi: REAL;
	rst: BOOL;
END_VAR
VAR_INPUT
END_VAR
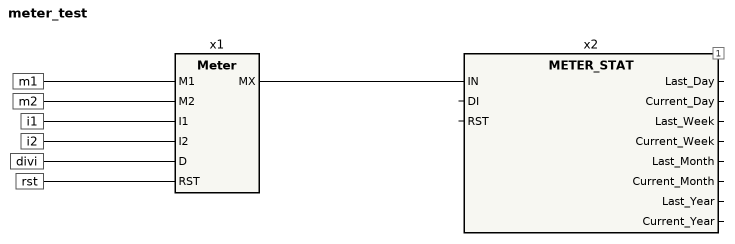
_CFC_ (* Continuous Function Chart, elements in execution order *)
#0 x1:Meter(M1: m1, M2: m2, I1: i1, I2: i2, D: divi, RST: rst)
#1 x2:METER_STAT(IN: #0.MX, DI: -, RST: -)
_END_CFC_
(* the same logic as Structured Text *)
x1(M1 := m1, M2 := m2, I1 := i1, I2 := i2, D := divi, RST := rst);
x2(IN := x1.MX);
END_PROGRAM

(* POU Engineering/measurements/Meter, ST *)
FUNCTION_BLOCK Meter
VAR_INPUT
	M1, M2 : REAL;
	I1, I2 : BOOL;
	D : REAL := 1;
	RST : BOOL;
END_VAR
VAR_OUTPUT RETAIN
	MX : REAL;
END_VAR
VAR
	int1 : FT_INT;
	int2 : FT_INT;
END_VAR

(*
	version 1.1	8. feb 2008
	programmer 	oscat
	tested BY		oscat

METER measures usage of power or similar values the output MX is the summ of the inputs over time.
MX := sum over time of I1 * P1 + I2 * P2.
a simple example is the consumption counter for a 2 stage oil burner where stage 1 is 10KW and stage 2 is 20KW.
I1 and I2 decide which value is accounted for, I1 = True only counts P1, I2 is True counts P2 
and I1 and I2 is true counts P1 and P2.
the meter can be used for all kind of consumption meters. P1 and P2 can change on the fly.

*)
(* meter would have a problem when int1 or int2 reach big values
and a short time tick would add a value smaller then the 7 digit resolution of real
therefore the variables m1 and m2 are used to store the counted values 
while the integrators are kept at small values to avoid this overrun
*)

int1(in := M1, Run := I1, rst := rst);
int2(in := M2, Run := I2, rst := rst);
MX := (int1.Out + int2.Out) / D;

(* revision history

hm	16. sep.2007		rev 1.0
	original version

hm	7. feb 2008		rev 1.1
	use new version of ft_int to avoid a counting stop at high values
	deleted unnecessary limits
*)
END_FUNCTION_BLOCK

(* POU Engineering/measurements/METER_STAT, ST *)
FUNCTION_BLOCK METER_STAT
VAR_INPUT
	IN : REAL;
	DI : DATE;
	RST : BOOL;
END_VAR
VAR_OUTPUT RETAIN
	Last_Day : REAL;
	Current_Day : REAL;
	Last_Week : REAL;
	Current_Week : REAL;
	Last_Month : REAL;
	Current_Month : REAL;
	Last_Year : REAL;
	Current_Year : REAL;
END_VAR
VAR RETAIN
	Year_Start : REAL;
	Month_Start : REAL;
	Week_Start : REAL;
	Day_Start : REAL;
	last_run: DATE;
END_VAR

(*
	version 1.0	16 sep 2007
	programmer 	oscat
	tested BY		oscat

METER_STAT runs statistics of a metered value, it calculates the current week, day, month and year consumption and stores the corresponding last day, week, month and year value.

*)
IF rst THEN
	Last_Day := 0;
	Current_Day := 0;
	Day_start := IN;
	Last_week := 0;
	Current_week := 0;
	Week_start := in;
	Last_month := 0;
	Current_month := 0;
	month_start := in;
	last_year := 0;
	current_year := 0;
	year_start := in;
ELSE
	Current_Day := IN - Day_Start;
	Current_Week := In - Week_Start;
	Current_Month := IN - Month_Start;
	Current_Year := IN - Year_Start;
END_IF;

IF year(DI) > year(last_run) THEN
	(* a new year has started *)
	last_year := current_year;
	current_year := 0;
	year_start := in;
	last_month := current_month;
	current_month := 0;
	month_start := in;
	last_day := current_day;
	current_day := 0;
	day_start := in;
ELSIF month(DI) > month(last_run) THEN
	(* a new month has started, january is alrerady done by year change *)
	last_month := current_month;
	current_month := 0;
	month_start := in;
	last_day := current_day;
	current_day := 0;
	day_start := in;
ELSIF day_of_year(di) > day_of_year(last_run) THEN
	(* day has chaged, first day of year and first day of month has already been taken care of *)
	last_day := current_day;
	current_day := 0;
	day_start := in;
END_IF;
IF weekday(DI) < weekday(last_run) THEN
	(* a new week has started *)
	last_week := current_week;
	current_week := 0;
	week_start := in;
END_IF;
last_run := di;

(* revision history
hm		16.9.2007		rev 1.0
	original version

*)
END_FUNCTION_BLOCK

(* POU XTEST/Baustein Tests/Net_com_test, CFC *)
PROGRAM Net_com_test
VAR
	X1: TCP_Client;
	x2: Net_Com;
	RBUF : ARRAY[0..Max_Receive_TCP_client] OF BYTE;
	error: BYTE;
	rdata: STRING(255);
END_VAR
VAR_INPUT
END_VAR
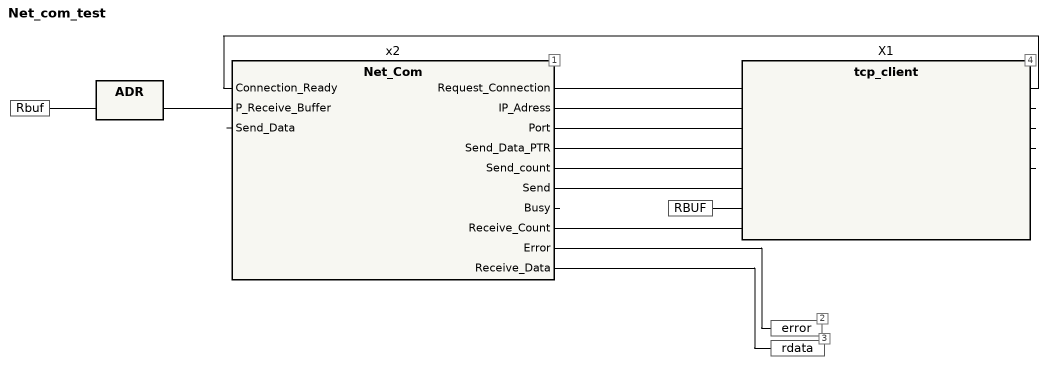
_CFC_ (* Continuous Function Chart, elements in execution order *)
#0 ADR(Rbuf)
#1 x2:Net_Com(Connection_Ready: #4.out 1, P_Receive_Buffer: #0, Send_Data: -, Server_IP := '85.214.80.110', Server_Port := 80)
#2 error <= #1.Error
#3 rdata <= #1.Receive_Data
#4 X1:tcp_client(#1.Request_Connection, #1.IP_Adress, #1.Port, #1.Send_Data_PTR, #1.Send_count, #1.Send, RBUF, #1.Receive_Count)
_END_CFC_
END_PROGRAM

(* POU XTEST/Ideas/Net_Com, ST *)
FUNCTION_BLOCK Net_Com
VAR_INPUT
	Connection_Ready : BOOL;
	P_Receive_Buffer : POINTER TO ARRAY[0..32000] OF BYTE;
	Send_Data : STRING(255) := 'GET / HTTP/1.1$R$NHost: www.oscat.de';

END_VAR
VAR_INPUT CONSTANT
	Server_IP : STRING(16);
	Server_Port : WORD := 80;
	Connect_timeout : TIME := T#3s;
	Transfer_timeout : TIME := T#3s;
END_VAR
VAR_OUTPUT
	Request_Connection : BOOL;
	IP_Adress : STRING(16);
	Port : WORD;
	Send_Data_PTR : POINTER TO ARRAY[0..32000] OF BYTE;
	Send_count : INT;
	Send : BOOL;
	Busy : BOOL;
	Receive_Count : DINT;
	Error : BYTE;
	Receive_Data : STRING(255);
END_VAR
VAR
	pts : POINTER TO ARRAY [0..32000] OF BYTE;
	i: INT;
	state: BYTE;
	stop: INT;
	tx: TIME;
	start: TIME;
END_VAR
(* read system time *)
tx := TIME();

CASE state OF
	0:	(* request connection if send_buffer contains data *)
		IF LEN(Send_Data) > 0 THEN
			error := 0;
			IP_adress := Server_IP;
			Port := Server_Port;
			request_connection := TRUE;
			state := 1;
			start := tx;
		END_IF;

	1:	(* connection was requested check for connection ready and transmit *)
		IF connection_ready THEN
			Send_count := LEN(Send_Data);
			Send_Data_ptr := ADR(Send_Data);
			Send := TRUE;
			state := 2;
		ELSIF tx - start >= connect_timeout THEN
			(* a connection was not established in time *)
			error := 10; (* connect timeout *)
			request_connection := FALSE;
			send_count := 0;
			Send_Data := '';
			state := 0;
		END_IF;

	2:	(* wait till server has returned an answer *)
		IF Receive_Count > 0 THEN
			IF receive_count > 254 THEN stop := 254; ELSE stop := DINT_TO_INT(receive_count); END_IF;
			Send := FALSE;
			request_connection := FALSE;
			(* copy bytes from receive_buffer to receive_data *)
			pts := ADR(Receive_Data);
			FOR I := 0 TO stop DO pts^[i] := P_receive_buffer^[i]; END_FOR;
			(* terminate the string with 0 *)
			pts^[i] := 0;
			(* clear receive_count and send buffer *)
			receive_count := 0;
			Send_Data := '';
			send_count := 0;
			state := 0;
		ELSIF tx - start >= transfer_timeout THEN
			error := 20; (* transfer timeout *)
			Send_Data := '';
			send_count := 0;
			request_connection := FALSE;
			send := FALSE;
			state := 0;
		END_IF;
END_CASE;

(*set the busy flag *)
busy := state > 0;
END_FUNCTION_BLOCK

(* POU XTEST/Performance Test/perf_test, CFC *)
PROGRAM perf_test
VAR
	x2: Performance;
	tc,tl8,tl32,ti,tf,ta: REAL;
	RSt: BOOL;
END_VAR
VAR_INPUT
END_VAR
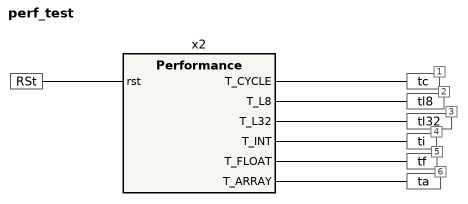
_CFC_ (* Continuous Function Chart, elements in execution order *)
#0 x2:Performance(rst: RSt)
#1 tc <= #0.T_CYCLE
#2 tl8 <= #0.T_L8
#3 tl32 <= #0.T_L32
#4 ti <= #0.T_INT
#5 tf <= #0.T_FLOAT
#6 ta <= #0.T_ARRAY
_END_CFC_
(* the same logic as Structured Text *)
x2(rst := RSt);
tc := x2.T_CYCLE;
tl8 := x2.T_L8;
tl32 := x2.T_L32;
ti := x2.T_INT;
tf := x2.T_FLOAT;
ta := x2.T_ARRAY;
END_PROGRAM

(* POU XTEST/Performance Test/Performance, ST *)
FUNCTION_BLOCK Performance
VAR_INPUT
	rst : BOOL;
END_VAR
VAR_OUTPUT
	T_CYCLE : REAL;
	T_L8 : REAL;
	T_L32 : REAL;
	T_INT : REAL;
	T_FLOAT : REAL;
	T_ARRAY : REAL;
END_VAR
VAR CONSTANT
	t_max : DWORD := 700;
	c_max : DWORD := 100000;
END_VAR
VAR
	mode : INT;
	start: DWORD;
	cycles : DWORD;
	tx: DWORD;
	init: BOOL;
END_VAR
IF rst OR NOT init THEN
	t_cycle := 1E10;
	t_l8 := 1E10;
	t_l32 := 1E10;
	t_int := 1E10;
	t_float := 1E10;
	t_array := 1E10;
	init := TRUE;
END_IF;
tx := T_PLC_MS();
CASE mode OF
0:	(* measure the execution time *)
	cycles := 0;
	mode := 1;
	start := tx;
1:	(* perform measurement for t_max *)
	IF (tx - start) < t_max THEN
		cycles := cycles + 1;
	ELSE
		T_cycle := MIN(DWORD_TO_REAL((tx - start) / cycles), t_cycle);
		mode := 2;
	END_IF;
2:	(* perform 8 Bit logic test *)
	start := tx;
	cycles := 0;
	REPEAT
		cycles := cycles + 1;
		TEST_L8();
	UNTIL (Cycles > C_max) OR ((T_PLC_MS() - start) >= t_max) END_REPEAT;
	T_L8 := MIN(DWORD_TO_REAL(T_PLC_MS() - start) / cycles, t_l8);
	mode := 3;
3:	(* perform 32 Bit logic test *)
	start := tx;
	cycles := 0;
	REPEAT
		cycles := cycles + 1;
		TEST_L32();
	UNTIL (Cycles > C_max) OR ((T_PLC_MS() - start) >= t_max) END_REPEAT;
	T_L32 := MIN(DWORD_TO_REAL(T_PLC_MS() - start) / cycles, T_L32);
	mode := 4;
4:	(* integer arithmetik Test *)
	start := tx;
	cycles := 0;
	REPEAT
		cycles := cycles + 1;
		TEST_INT();
	UNTIL (Cycles > C_max) OR ((T_PLC_MS() - start) >= t_max) END_REPEAT;
	T_INT := MIN(DWORD_TO_REAL(T_PLC_MS() - start) / cycles,T_INT);
	mode := 5;
5:	(* Floating Point Arithmetik test *)
	start := tx;
	cycles := 0;
	REPEAT
		cycles := cycles + 1;
		TEST_FLOAT();
	UNTIL (Cycles > C_max) OR ((T_PLC_MS() - start) >= t_max) END_REPEAT;
	T_FLOAT := MIN(DWORD_TO_REAL(T_PLC_MS() - start) / cycles,T_FLOAT);
	mode := 6;
6:	(* array sorting test *)
	start := tx;
	cycles := 0;
	REPEAT
		cycles := cycles + 1;
		TEST_ARRAY();
	UNTIL (Cycles > C_max) OR ((T_PLC_MS() - start) >= t_max) END_REPEAT;
	T_ARRAY := MIN(DWORD_TO_REAL(T_PLC_MS() - start) / cycles,T_ARRAY);
	mode := 0;
END_CASE;
END_FUNCTION_BLOCK

(* POU XTEST/Performance Test/TEST_L8, ST *)
FUNCTION TEST_L8 : BYTE
VAR_INPUT
END_VAR
VAR CONSTANT
	X : BYTE := 2#11110000;
	Y : BYTE := 2#01010101;
END_VAR
VAR
	i: INT;
END_VAR
FOR i := 1 TO 780 DO
	TEST_L8 := NOT(ROL(ROR(SHL(X XOR Y,4) AND SHR(X OR Y,4),4),3)) XOR Y AND X;
END_FOR;
END_FUNCTION

(* POU XTEST/Performance Test/TEST_L32, ST *)
FUNCTION TEST_L32 : DWORD
VAR_INPUT
END_VAR
VAR CONSTANT
	X : DWORD := 2#11110000_11111111_00000000_11110000;
	Y : DWORD := 2#01010101_00001111_11001100_00011100;
END_VAR
VAR
	i: INT;
END_VAR
FOR i := 1 TO 780 DO
	TEST_L32 := NOT(ROL(ROR(SHL(X XOR Y,12) AND SHR(X OR Y,13),14),13)) XOR Y AND X;
END_FOR;
END_FUNCTION

(* POU XTEST/Performance Test/TEST_INT, ST *)
FUNCTION TEST_INT : INT
VAR_INPUT
END_VAR
VAR CONSTANT
	X : INT := 21768;
	Y : INT := -657;
	Z : INT := 3;
END_VAR
VAR
	i: INT;
END_VAR
FOR i := 1 TO 790 DO
	TEST_INT := LIMIT(Y,ABS(DINT_TO_INT(Y * Y - Y +X) MOD Z)/(x-y),X) * Y -Z;
END_FOR;
END_FUNCTION

(* POU XTEST/Performance Test/TEST_FLOAT, ST *)
FUNCTION TEST_FLOAT : REAL
VAR_INPUT
END_VAR
VAR CONSTANT
	X : REAL := 3.1415;
	Y : REAL := 200000.23454;
END_VAR
VAR
	i: INT;
END_VAR
FOR i := 1 TO 405 DO
	TEST_FLOAT := EXP(LOG(TRUNC(LN(ABS((EXPT(y/X,X)-y+x)/Y)*COS(0.5)*SIN(0.5)*TAN(0.5)))*SQRT(X)));
END_FOR;
END_FUNCTION

(* POU XTEST/Performance Test/TEST_ARRAY, ST *)
FUNCTION TEST_ARRAY : BYTE
VAR_INPUT
END_VAR
VAR
	ta : ARRAY[0..7] OF REAL;
	i: INT;
END_VAR
FOR i := 1 TO 5 DO
	_array_sort(ADR(ta), SIZEOF(ta));
END_FOR;
END_FUNCTION

(* POU Mathematical/Array/_ARRAY_SORT, ST *)
FUNCTION _ARRAY_SORT : BOOL
VAR_INPUT
	f : POINTER TO ARRAY[1..32000] OF REAL;
	size : INT;
END_VAR
VAR
	i: INT;
	j: INT;
	temp : REAL;
	stop : INT;
	heapsize: INT;
	popmax : REAL;
	size2: INT;
	hs2: INT;
END_VAR

(*
version 1.5	5 jan 2008
programmer 	hugo
tested by		tobias

this function will sort a given array.
the function needs to be called:	_array_sort(adr("array"),sizeof("array"));
this function will manipulate a given array.
the function will not return anything except true, it will instead manipulate the original array.
because this function works with pointers its very time efficient and it needs no extra memory.

*)
(* generate heap *)

size := SHR(size,2);
size2 := SHR(size,1);
FOR i := SIZE2  TO 1 BY -1 DO 		(* zweite Hälfte des Feldes braucht nicht betrachtet werden *)
	j:=i;
    WHILE j <= SIZE2 DO
     	stop := j * 2 + 1;               (* finde Maximum der (beiden) Söhne *)
        IF stop > SIZE THEN stop := stop - 1;
        ELSIF f^[stop-1] > f^[stop] THEN stop := stop - 1;
		END_IF;
        IF f^[j] < f^[stop] THEN   		(* ggf. tauschen *)
         	temp := f^[j];
            f^[j] := f^[stop];
            f^[stop] := temp;
        END_IF;
        j := stop;
    END_WHILE;
END_FOR;

(* heapsort *)
FOR heapsize := size TO 1 BY -1 DO
	popmax := f^[1];
	f^[1] := f^[heapsize];
   	i := 1;
	hs2 := SHR(heapsize,1);
	WHILE i <= hs2 DO	     (* letztes Element an Anfang setzen und versickern lassen *)
       	stop := i * 2 + 1;                (* finde Maximum der (beiden) Söhne *)
        	IF stop > heapsize THEN stop := stop - 1;
        	ELSIF f^[stop-1] > f^[stop] THEN stop := stop - 1;
	 	END_IF;
        	IF f^[i] < f^[stop] THEN	     (* ggf. tauschen *)
            		temp := f^[i];
            		f^[i] := f^[stop];
            		f^[stop] := temp;
        	END_IF;
        	i := stop;
    	END_WHILE;
	f^[heapsize] := popmax;
END_FOR;

_array_sort := TRUE;

(* old algorithm bubble sort used before rev 1.2
stop := (size - SIZEOF(pt)) / SIZEOF(pt);
FOR i := 0 TO stop - 1 DO
	FOR m := i + 1 TO stop DO
		IF pt^[i] > pt^[m] THEN
			temp := pt^[i];
			pt^[i] := pt^[m];
			pt^[m] := temp;
		END_IF;
	END_FOR;
END_FOR;
_array_sort := TRUE;

*)
(* revision history

hm 	6.1.2007 	rev 1.1
	changed return value to true

hm	22. sep 2007	rev 1.2
	changed sorting algorithm to heap sort for performance reasons

hm 	14. nov 2007	rev 1.3
	changed calculation of stop to be more efficient

hm	15 dec 2007		rev 1.4
	added function return true

hm	5. jan 2008		rev 1.5
	improved performance
*)
END_FUNCTION

(* POU XTEST/Baustein Tests/reverse_test, CFC *)
PROGRAM reverse_test
VAR
	s1: STRING;
	in: BYTE;
END_VAR
VAR_INPUT
END_VAR
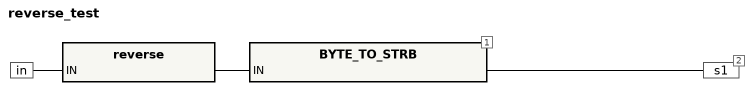
_CFC_ (* Continuous Function Chart, elements in execution order *)
#0 reverse(IN: in)
#1 BYTE_TO_STRB(IN: #0)
#2 s1 <= #1
_END_CFC_
(* the same logic as Structured Text *)
s1 := BYTE_TO_STRB(IN := reverse(IN := in));
END_PROGRAM

(* POU XTEST/Baustein Tests/rmp_test, CFC *)
PROGRAM rmp_test
VAR
	set, rst, en, ud : BOOL;
	y : BYTE;
	bsy, on, off : BOOL;
	y1 : WORD;
	bsy1, on1, off1 : BOOL;
	x1: rmp_B;
	x2 : rmp_W;
	x3 : rmp_W;
	x6: RS;
	x4: TP;
	x5: TP;
	x7: rmp_B;
	rmp2: BYTE;
	bsy2: BOOL;
	bsy0: BOOL;
	ramp0: WORD;
	x8: m_t;
	tt: TIME;
	x9: m_t;
	t1: TIME;
	x10: m_t;
	t2: TIME;
END_VAR
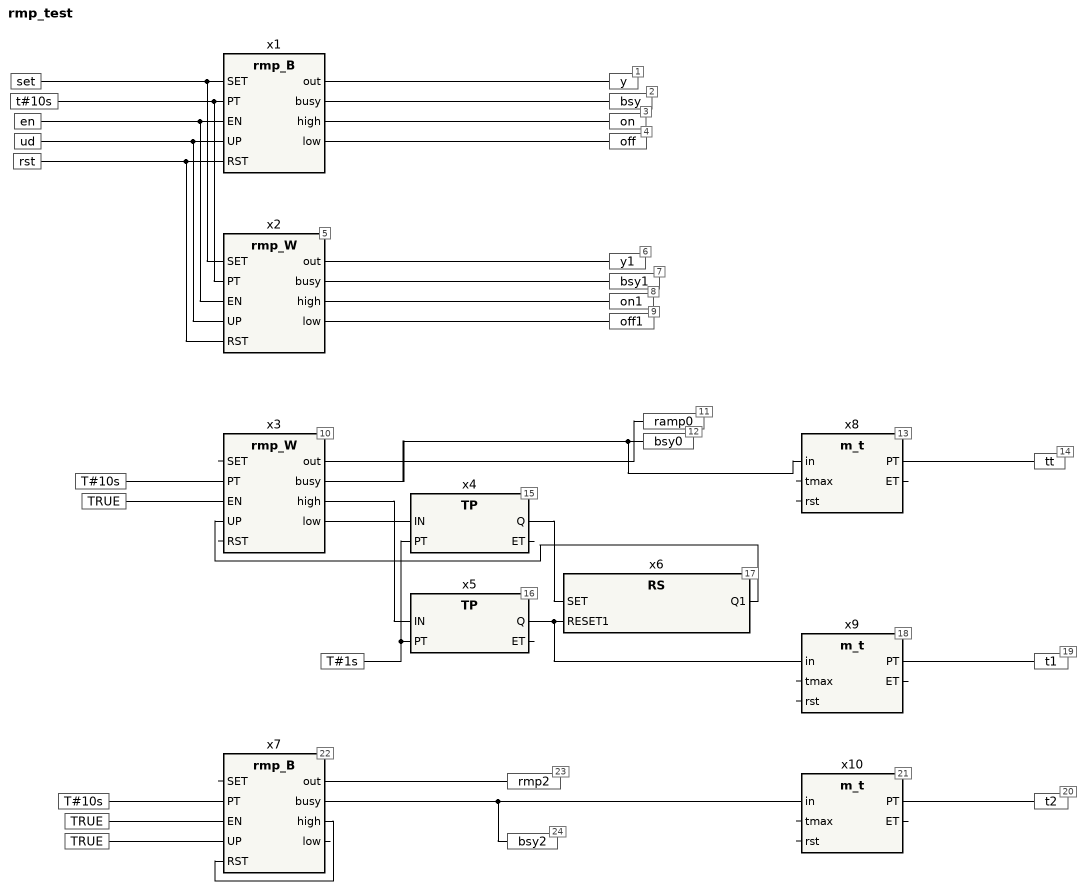
_CFC_ (* Continuous Function Chart, elements in execution order *)
#0 x1:rmp_B(SET: set, PT: t#10s, EN: en, UP: ud, RST: rst)
#1 y <= #0.out
#2 bsy <= #0.busy
#3 on <= #0.high
#4 off <= #0.low
#5 x2:rmp_W(SET: set, PT: t#10s, EN: en, UP: ud, RST: rst)
#6 y1 <= #5.out
#7 bsy1 <= #5.busy
#8 on1 <= #5.high
#9 off1 <= #5.low
#10 x3:rmp_W(SET: -, PT: T#10s, EN: TRUE, UP: #17.Q1, RST: -)
#11 ramp0 <= #10.out
#12 bsy0 <= #10.busy
#13 x8:m_t(in: #10.busy, tmax: -, rst: -)
#14 tt <= #13.PT
#15 x4:TP(IN: #10.low, PT: T#1s)
#16 x5:TP(IN: #10.high, PT: T#1s)
#17 x6:RS(SET: #15.Q, RESET1: #16.Q)
#18 x9:m_t(in: #16.Q, tmax: -, rst: -)
#19 t1 <= #18.PT
#20 t2 <= #21.PT
#21 x10:m_t(in: #22.busy, tmax: -, rst: -)
#22 x7:rmp_B(SET: -, PT: T#10s, EN: TRUE, UP: TRUE, RST: #22.high)
#23 rmp2 <= #22.out
#24 bsy2 <= #22.busy
_END_CFC_
(* the same logic as Structured Text *)
x1(SET := set, PT := t#10s, EN := en, UP := ud, RST := rst);
y := x1.out;
bsy := x1.busy;
on := x1.high;
off := x1.low;
x2(SET := set, PT := t#10s, EN := en, UP := ud, RST := rst);
y1 := x2.out;
bsy1 := x2.busy;
on1 := x2.high;
off1 := x2.low;
x3(PT := T#10s, EN := TRUE, UP := x6.Q1);
ramp0 := x3.out;
bsy0 := x3.busy;
x8(in := x3.busy);
tt := x8.PT;
x4(IN := x3.low, PT := T#1s);
x5(IN := x3.high, PT := T#1s);
x6(SET := x4.Q, RESET1 := x5.Q);
x9(in := x5.Q);
t1 := x9.PT;
t2 := x10.PT;
x10(in := x7.busy);
x7(PT := T#10s, EN := TRUE, UP := TRUE, RST := x7.high);
rmp2 := x7.out;
bsy2 := x7.busy;
END_PROGRAM

(* POU Engineering/signal generators/rmp_W, ST *)
FUNCTION_BLOCK rmp_W
VAR_INPUT
	SET : BOOL := FALSE;
	PT : TIME;
	EN : BOOL := TRUE;
	UP : BOOL := TRUE;
	RST : BOOL := FALSE;
END_VAR
VAR_OUTPUT
	out : WORD;
	busy : BOOL;
	high : BOOL;
	low : BOOL;
END_VAR
VAR CONSTANT
	FF : WORD := 65535;
END_VAR
VAR
	last_step : DWORD;
	now : DWORD;
	tmp: DWORD;
	edge: BOOL;
	N: WORD;
	init: BOOL;
END_VAR

(*
	version 1.7	25. dec 2007
	programmer 	oscat
	tested BY		oscat

this ramp generator generates a Word wide ramp with 65535 steps
the generator has an asynchronous set and reset
the ramp is controlled by PT which is the total ramp time for a full sweep from 0..65535
an UD input controlls the direction Up or Down and the E input enables the ramp generation
a busy output indicates that the ramp is running, busy false means output is stable.
the outputs low and high will be true when the output has reached its max or min value.
*)
(* read system time *)
now := T_PLC_MS();

(* init code for startup *)
IF NOT init THEN
	init := TRUE;
	last_step := now;
END_IF;

(* calculate the necessary step response *)
IF pt = t#0s THEN
	tmp := FF;
ELSE
	tmp := SHL(now - last_step, 16) / TIME_TO_DWORD(pt);
END_IF;
IF tmp > FF THEN N:= FF; ELSE N:= DWORD_TO_WORD(tmp); END_IF;

(* detetct edge on en *)
IF en AND NOT edge THEN
	last_step := now;
(* check for asynchronous set or reset *)
ELSIF rst THEN
	out := 0;
ELSIF set  THEN
	out := FF;
ELSIF en THEN
	(* generate ramp *)
	last_step := now;
	IF UP THEN
		IF out > FF - N THEN out := FF; ELSE out := out + N; END_IF;
	ELSE
		IF out < N THEN out := 0; ELSE out := out - N; END_IF;
	END_IF;
END_IF;
edge := en;

(* checks for outputs stable and reset or set busy flag *)
IF out = 0 THEN
	busy := FALSE;
	low := TRUE;
	high := FALSE;
ELSIF out = FF THEN
	busy := FALSE;
	high := TRUE;
	low := FALSE;
ELSE
	busy := en;
	high := FALSE;
	low := FALSE;
END_IF;

(* revision history:

hm 4.10.2006		rev 1.1
	added the busy output which signals that the ramp is running.

hm 22.1.2007		rev 1.2
	deleted unused variable step

hm	17.9.2007		rev 1.3
	replaced time() with t_plc_ms() for compatibility reasons

hm	28. sep 2007	rev 1.4
	added outputs on and off
	busy is now disabled while en is false
	new coding for higher accuracy and performance

hm	5. oct 2007		rev 1.5
	added statements to allow for PT to be t#0s output jumps to max or min immediately

hm	2. dec 2007		rev 1.6
	corrected an error in calculation of step response

hm	25. dec 2007	rev 1.7
	corrected an error while step response was too slow for fast rise times
*)
END_FUNCTION_BLOCK

(* POU Engineering/measurements/m_t, ST *)
FUNCTION_BLOCK m_t
VAR_INPUT
	in: BOOL;
	tmax : TIME := t#10d;
	rst: BOOL;
END_VAR
VAR_OUTPUT
	PT : TIME := t#0ms;
	ET: TIME;
END_VAR
VAR
	edge : BOOL := 0;
	start : TIME;
	stop : TIME;
	init : BOOL;
	tx: TIME;
	startup: BOOL;
END_VAR

(*
	version 1.2	16 sep 2007
	programmer 	hugo
	tested BY		tobias

m_t measures the with of a high pulse and returs the last measured pulse width on output PT.
a second output ET is starting from 0 at the rising edge and counting up until the falling edge occurs and resetts et to 0.
the asynchrtonous input rst can reset the outputs at any time.
tmax defines a maximum measurable time, if this value is exceeded the outputs will be reset to 0.
*)
(* check for rst input *)
IF rst OR et >= tmax THEN
	init := FALSE;
	startup := FALSE;
	pt := t#0ms;
	et := t#0ms;
END_IF;

(* avoid timers to start when input is true at startup *)
IF NOT startup THEN
	edge := in;
	startup := TRUE;
END_IF;

(* read system timer *)
tx := DWORD_TO_TIME(T_PLC_MS());

(* edge trigger rising and falling edge *)
IF in XOR edge THEN
	edge := in;
	(* rising edge starts measurement *)
	IF in THEN
		init := TRUE;
		start := Tx;
	(* falling edge stops measurement *)
	ELSIF init THEN
		stop := Tx;
		pt := stop - start;
	END_IF;
END_IF;

IF init AND in THEN
	et := Tx - start; ELSE et := t#0ms;
END_IF;

(* revision history
hm		4.8.2006	rev 1.0
	original version

hm		2.5.2007	rev 1.1
	added init variable to avoid unreasonable measurement if falling edge occurs first.
	added et (elapsed time) output to count from 0 at rising edge until a falling edge resets et to 0.
	added reset input.

hm		16.9.2007	rev 1.2
	changes time() to T_plc_ms() for compatibility reasons

*)
END_FUNCTION_BLOCK

(* POU XTEST/Baustein Tests/sensor_test, CFC *)
PROGRAM sensor_test
VAR
	t: REAL;
	tn: REAL;
	tm: REAL;
	ts: REAL;
	dtn: REAL;
	fp: REAL;
END_VAR
VAR_INPUT
END_VAR
VAR (* helpers for the ST form of the networks *)
	_t290 : REAL;
	_t339 : REAL;
END_VAR
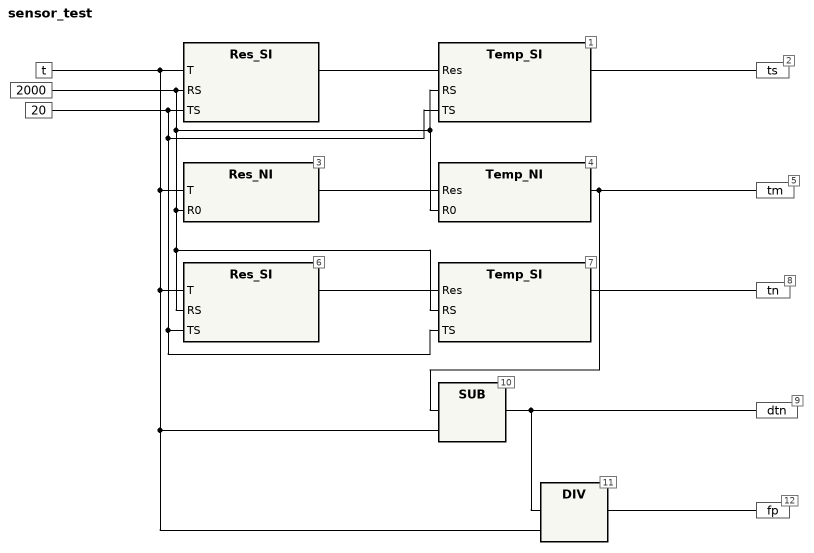
_CFC_ (* Continuous Function Chart, elements in execution order *)
#0 Res_SI(T: t, RS: 2000, TS: 20)
#1 Temp_SI(Res: #0, RS: 2000, TS: 20)
#2 ts <= #1
#3 Res_NI(T: t, R0: 2000)
#4 Temp_NI(Res: #3, R0: 2000)
#5 tm <= #4
#6 Res_SI(T: t, RS: 2000, TS: 20)
#7 Temp_SI(Res: #6, RS: 2000, TS: 20)
#8 tn <= #7
#9 dtn <= #10
#10 SUB(#4, t)
#11 DIV(#10, t)
#12 fp <= #11
_END_CFC_
(* the same logic as Structured Text *)
ts := Temp_SI(Res := Res_SI(T := t, RS := 2000, TS := 20), RS := 2000, TS := 20);
_t290 := Temp_NI(Res := Res_NI(T := t, R0 := 2000), R0 := 2000);
tm := _t290;
tn := Temp_SI(Res := Res_SI(T := t, RS := 2000, TS := 20), RS := 2000, TS := 20);
dtn := _t339;
_t339 := _t290 - t;
fp := _t339 / t;
END_PROGRAM

(* POU Engineering/sensor/Res_SI, ST *)
FUNCTION Res_SI : REAL
VAR_INPUT
	T : REAL;
	RS : REAL;
	TS : REAL;
END_VAR
VAR CONSTANT
	A : REAL := 7.64E-3;
	B : REAL := 1.66E-5;
END_VAR
VAR
	TX: REAL;
END_VAR

(*
version 1.1	2 dec 2007
programmer 	hugo
tested by		tobias

this function returs the resistance for a silicon sensor for a temperature range from -50..+150 °C
for example KTY10 normaly Rs at 25 °C
*)
TX := T - TS;
Res_SI := RS * ( 1 + A * TX + B * TX * TX);

(* revision history
hm		4. aug 2006		rev 1.0
	original version

hm		2. dec 2007		rev 1.1
	changed code for better performance

*)
END_FUNCTION

(* POU Engineering/sensor/Temp_SI, ST *)
FUNCTION Temp_SI : REAL
VAR_INPUT
	Res : REAL;
	RS : REAL;
	TS : REAL;
END_VAR
VAR CONSTANT
END_VAR
VAR
END_VAR

(*
version 1.4	6. jan 2008
programmer 	hugo
tested by		tobias

this function returs the temperature for a silicon sensor for a range from -60..+180 °C
for example KTY10 RS at TS normally 25 °C
*)
Temp_SI := (-7.64E-3 + SQRT(Res/RS* 6.64E-5 - 0.803E-5)) * 30120.48193 + TS;

(* code before rev 1.3
Temp_SI := -60;
WHILE step > accuracy DO
	(* test if result greater or less *)
	IF Res_SI(Temp_SI + step,RS,TS) < Res THEN Temp_SI := Temp_SI + step; END_IF;
	step := step / 2;
END_WHILE;
*)

(* revision history

hm 24.1.2007		rev 1.1
	the function would only work for TS = 25, now it works for other values of ts.

hm 10.9.2007		rev 1.2
	changed the function to use successive approcimation to avoid an error generated by a sqrt from a negative result.
	changed accuracy to 0.02 degrees to shorten execution time

hm 17. 12 2007		rev 1.3
	improovements for better performance

hm	6. jan 2008		rev 1.4
	further performance improvement
*)
END_FUNCTION

(* POU Engineering/sensor/Res_NI, ST *)
FUNCTION Res_NI : REAL
VAR_INPUT
	T : REAL;
	R0 : REAL;
END_VAR
VAR CONSTANT
	A : REAL := 0.5485;
	B : REAL := 0.665E-3;
	C : REAL := 2.805E-9;
END_VAR
VAR
	T2: REAL;
END_VAR

(*
version 1.2	2 dec 2007
programmer 	hugo
tested by		tobias

this function returs the resistance for a nickel sensor for a temperature range from -60..+180 °C *)
T2 := T*T;
Res_NI := R0 + A*T + B*T2 + C*T2*T2;

(* revision history

hm	4.8.2006		rev 1.0
	original version

hm	13.9.2007		rev 1.1
	changed coding for better performance

hm	2. dec. 2007	rev 1.2
	changed code for better performance
*)

(*

 Auszug aus DIN 43760 für Ni100

°C		R		°C		R		°C	R		°C		R		°C		R

-60 	69,5 	-10 	94,6 	40 	123,0 	90 		154,9 	140 	190,9
-55 	71,9 	-5 		97,3 	45 	126,0 	95 		158,3 	145 	194,8
-50 	74,3 	0 		100,0 	50 	129,1 	100 	161,8 	150 	198,7
-45 	76,7 	5 		102,8 	55 	132,2 	105 	165,3 	155 	202,6
-40 	79,1 	10 		105,6 	60 	135,3 	110 	168,8 	160 	206,6
-35 	81,6 	15 		108,4 	65 	138,5 	115 	172,4 	165 	210,7
-30 	84,2 	20 		111,2 	70 	141,7 	120 	176,0 	170 	214,8
-25 	86,7 	25 		114,1 	75 	145,0 	125 	179,6 	175 	219,0
-20 	89,3 	30 		117,1 	80 	148,3 	130 	183,3 	180 	223,2
-15 	91,9 	35 		120,0 	85 	151,6 	135 	187,1 	  	 

*)
END_FUNCTION

